   // // TIF[10].FixedLoc : Tool fixed location coded / Emplacement fixe d'outil codé
   // // TIF[11].FixedLoc : Tool fixed location coded / Emplacement fixe d'outil codé
   // // TIF[12].FixedLoc : Tool fixed location coded / Emplacement fixe d'outil codé
   // // TIF[13].FixedLoc : Tool fixed location coded / Emplacement fixe d'outil codé
   // // TIF[14].FixedLoc : Tool fixed location coded / Emplacement fixe d'outil codé
   // // TIF[15].FixedLoc : Tool fixed location coded / Emplacement fixe d'outil codé
   // // TIF[16].FixedLoc : Tool fixed location coded / Emplacement fixe d'outil codé
   // // TIF[2].Used : Tool was in use / Outil a été utilisé
   // // TIF[3].Used : Tool was in use / Outil a été utilisé
   // // TIF[4].Used : Tool was in use / Outil a été utilisé
   // // TIF[5].Used : Tool was in use / Outil a été utilisé
   // // TIF[6].Used : Tool was in use / Outil a été utilisé
   // // TIF[7].Used : Tool was in use / Outil a été utilisé
   // // TIF[8].Used : Tool was in use / Outil a été utilisé
   // // TIF[9].Used : Tool was in use / Outil a été utilisé
   // // TIF[10].Used : Tool was in use / Outil a été utilisé
   // // TIF[11].Used : Tool was in use / Outil a été utilisé
   // // TIF[12].Used : Tool was in use / Outil a été utilisé
   // // TIF[13].Used : Tool was in use / Outil a été utilisé
   // // TIF[14].Used : Tool was in use / Outil a été utilisé
   // // TIF[15].Used : Tool was in use / Outil a été utilisé
   // // TIF[16].Used : Tool was in use / Outil a été utilisé
   // // TIF[2].TNo : Tool new: T number / Nouvel outil : numéro d'outil
   // // TIF[3].TNo : Tool new: T number / Nouvel outil : numéro d'outil
   // // TIF[4].TNo : Tool new: T number / Nouvel outil : numéro d'outil
   // // TIF[5].TNo : Tool new: T number / Nouvel outil : numéro d'outil
   // // TIF[6].TNo : Tool new: T number / Nouvel outil : numéro d'outil
   // // TIF[7].TNo : Tool new: T number / Nouvel outil : numéro d'outil
   // // TIF[8].TNo : Tool new: T number / Nouvel outil : numéro d'outil
   // // TIF[9].TNo : Tool new: T number / Nouvel outil : numéro d'outil
   // // TIF[10].TNo : Tool new: T number / Nouvel outil : numéro d'outil
   // // TIF[11].TNo : Tool new: T number / Nouvel outil : numéro d'outil
   // // TIF[12].TNo : Tool new: T number / Nouvel outil : numéro d'outil
   // // TIF[13].TNo : Tool new: T number / Nouvel outil : numéro d'outil
   // // TIF[14].TNo : Tool new: T number / Nouvel outil : numéro d'outil
   // // TIF[15].TNo : Tool new: T number / Nouvel outil : numéro d'outil
   // // TIF[16].TNo : Tool new: T number / Nouvel outil : numéro d'outil
   // // TIF[2].MyPlace : Original location of new tool / Emplacement d'origine du nouvel outil
   // // TIF[3].MyPlace : Original location of new tool / Emplacement d'origine du nouvel outil
   // // TIF[4].MyPlace : Original location of new tool / Emplacement d'origine du nouvel outil
   // // TIF[5].MyPlace : Original location of new tool / Emplacement d'origine du nouvel outil
   // // TIF[6].MyPlace : Original location of new tool / Emplacement d'origine du nouvel outil
   // // TIF[7].MyPlace : Original location of new tool / Emplacement d'origine du nouvel outil
   // // TIF[8].MyPlace : Original location of new tool / Emplacement d'origine du nouvel outil
   // // TIF[9].MyPlace : Original location of new tool / Emplacement d'origine du nouvel outil
   // // TIF[10].MyPlace : Original location of new tool / Emplacement d'origine du nouvel outil
   // // TIF[11].MyPlace : Original location of new tool / Emplacement d'origine du nouvel outil
   // // TIF[12].MyPlace : Original location of new tool / Emplacement d'origine du nouvel outil
   // // TIF[13].MyPlace : Original location of new tool / Emplacement d'origine du nouvel outil
   // // TIF[14].MyPlace : Original location of new tool / Emplacement d'origine du nouvel outil
   // // TIF[15].MyPlace : Original location of new tool / Emplacement d'origine du nouvel outil
   // // TIF[16].MyPlace : Original location of new tool / Emplacement d'origine du nouvel outil
END_TYPE

TYPE "LBP_typeTMTurretMT"
TITLE = Tool management / Gestion des outils
// User data type for block LBP_TMTurretMT [DB1073] / Type de données utilisateur pour bloc LBP_TMTurretMT [DB1073]
   STRUCT
      MTIF : Array[1..16] of Struct
         DistanceCoding : Int;   // Type of distance coding ($TC_MTP_KD) / Type de codage de distance ($TC_MTP_KD)
         Places : Int;   // Number of locations of the multitool / Nombre d'emplacements Multitool
         Distance : Real;   // Multitool location distance / Distance de l'emplacement Multitool
         NewMTNo : Int;   // MT-Number new Tool / Numéro MT du nouvel outil
         NewPlace : Int;   // Multitool place number / Numéro d'emplacement Multitool
         OldMTNo : Int;   // MT-Number old Tool / Numéro MT de l'ancien outil
         OldPlace : Int;   // Multitool place number / Numéro d'emplacement Multitool
         LocType : Int;   // Tool new: location type / Nouvel outil : type d'emplacement
         SLeft : Int;   // Tool new: size left / Nouvel outil : taille côté gauche
         SRight : Int;   // Tool new: size right / Nouvel outil : taille côté droit
         STop : Int;   // Tool new: size top / Nouvel outil : taille dessus
         SBottom : Int;   // Tool new: size bottom / Nouvel outil : taille dessous
         TInBuffer : Bool;   // ID for tools in buffer / ID pour outils dans tampon
         IgnoreDisabled : Bool;   // Ignore disabled / Ignorer désactivation
         Unload : Bool;   // To be unloaded / À décharger
         Load : Bool;   // To be loaded / À charger
         MasterTool : Bool;   // Tool is the master tool / L'outil est un outil principal
         n26_5 : Bool;   // Reserved / Réservé
         n26_6 : Bool;   // Reserved / Réservé
         HandTool : Bool;   // Hand tool / Outil manuel
         Active : Bool;   // Active tool / Outil actif
         Enabled : Bool;   // Tool enabled / Outil activé
         Disabled : Bool;   // Tool disabled / Outil désactivé
         Measured : Bool;   // Tool measured / Outil mesuré
         Prewarn : Bool;   // Prewarning limit reached / Seuil de préavis atteint
         Change : Bool;   // Tool being changed / Outil en cours de changement
         FixedLoc : Bool;   // Tool fixed location coded / Emplacement fixe d'outil codé
         Used : Bool;   // Tool was in use / Outil a été utilisé
         TNo : Int;   // Tool new: T number / Nouvel outil : numéro d'outil
         Toolholder : Int;   // Toolholder number as tool compensation reference / Numéro de porte-outil en tant que référence pour la compensation d'outil
         MyMag : Int;   // Multitool number the tool is loaded onto / Numéro Multitool dans lequel l'outil est chargé
         MyPlace : Int;   // Multitool place number / Numéro d'emplacement Multitool
         reserved : Array[1..7] of Int;   // Reserved / Réservé
      END_STRUCT;
   END_STRUCT;
   // // MTIF[2].DistanceCoding : Type of distance coding ($TC_MTP_KD) / Type de codage de distance ($TC_MTP_KD)
   // // MTIF[3].DistanceCoding : Type of distance coding ($TC_MTP_KD) / Type de codage de distance ($TC_MTP_KD)
   // // MTIF[4].DistanceCoding : Type of distance coding ($TC_MTP_KD) / Type de codage de distance ($TC_MTP_KD)
   // // MTIF[5].DistanceCoding : Type of distance coding ($TC_MTP_KD) / Type de codage de distance ($TC_MTP_KD)
   // // MTIF[6].DistanceCoding : Type of distance coding ($TC_MTP_KD) / Type de codage de distance ($TC_MTP_KD)
   // // MTIF[7].DistanceCoding : Type of distance coding ($TC_MTP_KD) / Type de codage de distance ($TC_MTP_KD)
   // // MTIF[8].DistanceCoding : Type of distance coding ($TC_MTP_KD) / Type de codage de distance ($TC_MTP_KD)
   // // MTIF[9].DistanceCoding : Type of distance coding ($TC_MTP_KD) / Type de codage de distance ($TC_MTP_KD)
   // // MTIF[10].DistanceCoding : Type of distance coding ($TC_MTP_KD) / Type de codage de distance ($TC_MTP_KD)
   // // MTIF[11].DistanceCoding : Type of distance coding ($TC_MTP_KD) / Type de codage de distance ($TC_MTP_KD)
   // // MTIF[12].DistanceCoding : Type of distance coding ($TC_MTP_KD) / Type de codage de distance ($TC_MTP_KD)
   // // MTIF[13].DistanceCoding : Type of distance coding ($TC_MTP_KD) / Type de codage de distance ($TC_MTP_KD)
   // // MTIF[14].DistanceCoding : Type of distance coding ($TC_MTP_KD) / Type de codage de distance ($TC_MTP_KD)
   // // MTIF[15].DistanceCoding : Type of distance coding ($TC_MTP_KD) / Type de codage de distance ($TC_MTP_KD)
   // // MTIF[16].DistanceCoding : Type of distance coding ($TC_MTP_KD) / Type de codage de distance ($TC_MTP_KD)
   // // MTIF[2].Places : Number of locations of the multitool / Nombre d'emplacements Multitool
   // // MTIF[3].Places : Number of locations of the multitool / Nombre d'emplacements Multitool
   // // MTIF[4].Places : Number of locations of the multitool / Nombre d'emplacements Multitool
   // // MTIF[5].Places : Number of locations of the multitool / Nombre d'emplacements Multitool
   // // MTIF[6].Places : Number of locations of the multitool / Nombre d'emplacements Multitool
   // // MTIF[7].Places : Number of locations of the multitool / Nombre d'emplacements Multitool
   // // MTIF[8].Places : Number of locations of the multitool / Nombre d'emplacements Multitool
   // // MTIF[9].Places : Number of locations of the multitool / Nombre d'emplacements Multitool
   // // MTIF[10].Places : Number of locations of the multitool / Nombre d'emplacements Multitool
   // // MTIF[11].Places : Number of locations of the multitool / Nombre d'emplacements Multitool
   // // MTIF[12].Places : Number of locations of the multitool / Nombre d'emplacements Multitool
   // // MTIF[13].Places : Number of locations of the multitool / Nombre d'emplacements Multitool
   // // MTIF[14].Places : Number of locations of the multitool / Nombre d'emplacements Multitool
   // // MTIF[15].Places : Number of locations of the multitool / Nombre d'emplacements Multitool
   // // MTIF[16].Places : Number of locations of the multitool / Nombre d'emplacements Multitool
   // // MTIF[2].Distance : Multitool location distance / Distance de l'emplacement Multitool
   // // MTIF[3].Distance : Multitool location distance / Distance de l'emplacement Multitool
   // // MTIF[4].Distance : Multitool location distance / Distance de l'emplacement Multitool
   // // MTIF[5].Distance : Multitool location distance / Distance de l'emplacement Multitool
   // // MTIF[6].Distance : Multitool location distance / Distance de l'emplacement Multitool
   // // MTIF[7].Distance : Multitool location distance / Distance de l'emplacement Multitool
   // // MTIF[8].Distance : Multitool location distance / Distance de l'emplacement Multitool
   // // MTIF[9].Distance : Multitool location distance / Distance de l'emplacement Multitool
   // // MTIF[10].Distance : Multitool location distance / Distance de l'emplacement Multitool
   // // MTIF[11].Distance : Multitool location distance / Distance de l'emplacement Multitool
   // // MTIF[12].Distance : Multitool location distance / Distance de l'emplacement Multitool
   // // MTIF[13].Distance : Multitool location distance / Distance de l'emplacement Multitool
   // // MTIF[14].Distance : Multitool location distance / Distance de l'emplacement Multitool
   // // MTIF[15].Distance : Multitool location distance / Distance de l'emplacement Multitool
   // // MTIF[16].Distance : Multitool location distance / Distance de l'emplacement Multitool
   // // MTIF[2].NewMTNo : MT-Number new Tool / Numéro MT du nouvel outil
   // // MTIF[3].NewMTNo : MT-Number new Tool / Numéro MT du nouvel outil
   // // MTIF[4].NewMTNo : MT-Number new Tool / Numéro MT du nouvel outil
   // // MTIF[5].NewMTNo : MT-Number new Tool / Numéro MT du nouvel outil
   // // MTIF[6].NewMTNo : MT-Number new Tool / Numéro MT du nouvel outil
   // // MTIF[7].NewMTNo : MT-Number new Tool / Numéro MT du nouvel outil
   // // MTIF[8].NewMTNo : MT-Number new Tool / Numéro MT du nouvel outil
   // // MTIF[9].NewMTNo : MT-Number new Tool / Numéro MT du nouvel outil
   // // MTIF[10].NewMTNo : MT-Number new Tool / Numéro MT du nouvel outil
   // // MTIF[11].NewMTNo : MT-Number new Tool / Numéro MT du nouvel outil
   // // MTIF[12].NewMTNo : MT-Number new Tool / Numéro MT du nouvel outil
   // // MTIF[13].NewMTNo : MT-Number new Tool / Numéro MT du nouvel outil
   // // MTIF[14].NewMTNo : MT-Number new Tool / Numéro MT du nouvel outil
   // // MTIF[15].NewMTNo : MT-Number new Tool / Numéro MT du nouvel outil
   // // MTIF[16].NewMTNo : MT-Number new Tool / Numéro MT du nouvel outil
   // // MTIF[2].NewPlace : Multitool place number / Numéro d'emplacement Multitool
   // // MTIF[3].NewPlace : Multitool place number / Numéro d'emplacement Multitool
   // // MTIF[4].NewPlace : Multitool place number / Numéro d'emplacement Multitool
   // // MTIF[5].NewPlace : Multitool place number / Numéro d'emplacement Multitool
   // // MTIF[6].NewPlace : Multitool place number / Numéro d'emplacement Multitool
   // // MTIF[7].NewPlace : Multitool place number / Numéro d'emplacement Multitool
   // // MTIF[8].NewPlace : Multitool place number / Numéro d'emplacement Multitool
   // // MTIF[9].NewPlace : Multitool place number / Numéro d'emplacement Multitool
   // // MTIF[10].NewPlace : Multitool place number / Numéro d'emplacement Multitool
   // // MTIF[11].NewPlace : Multitool place number / Numéro d'emplacement Multitool
   // // MTIF[12].NewPlace : Multitool place number / Numéro d'emplacement Multitool
   // // MTIF[13].NewPlace : Multitool place number / Numéro d'emplacement Multitool
   // // MTIF[14].NewPlace : Multitool place number / Numéro d'emplacement Multitool
   // // MTIF[15].NewPlace : Multitool place number / Numéro d'emplacement Multitool
   // // MTIF[16].NewPlace : Multitool place number / Numéro d'emplacement Multitool
   // // MTIF[2].OldMTNo : MT-Number old Tool / Numéro MT de l'ancien outil
   // // MTIF[3].OldMTNo : MT-Number old Tool / Numéro MT de l'ancien outil
   // // MTIF[4].OldMTNo : MT-Number old Tool / Numéro MT de l'ancien outil
   // // MTIF[5].OldMTNo : MT-Number old Tool / Numéro MT de l'ancien outil
   // // MTIF[6].OldMTNo : MT-Number old Tool / Numéro MT de l'ancien outil
   // // MTIF[7].OldMTNo : MT-Number old Tool / Numéro MT de l'ancien outil
   // // MTIF[8].OldMTNo : MT-Number old Tool / Numéro MT de l'ancien outil
   // // MTIF[9].OldMTNo : MT-Number old Tool / Numéro MT de l'ancien outil
   // // MTIF[10].OldMTNo : MT-Number old Tool / Numéro MT de l'ancien outil
   // // MTIF[11].OldMTNo : MT-Number old Tool / Numéro MT de l'ancien outil
   // // MTIF[12].OldMTNo : MT-Number old Tool / Numéro MT de l'ancien outil
   // // MTIF[13].OldMTNo : MT-Number old Tool / Numéro MT de l'ancien outil
   // // MTIF[14].OldMTNo : MT-Number old Tool / Numéro MT de l'ancien outil
   // // MTIF[15].OldMTNo : MT-Number old Tool / Numéro MT de l'ancien outil
   // // MTIF[16].OldMTNo : MT-Number old Tool / Numéro MT de l'ancien outil
   // // MTIF[2].OldPlace : Multitool place number / Numéro d'emplacement Multitool
   // // MTIF[3].OldPlace : Multitool place number / Numéro d'emplacement Multitool
   // // MTIF[4].OldPlace : Multitool place number / Numéro d'emplacement Multitool
   // // MTIF[5].OldPlace : Multitool place number / Numéro d'emplacement Multitool
   // // MTIF[6].OldPlace : Multitool place number / Numéro d'emplacement Multitool
   // // MTIF[7].OldPlace : Multitool place number / Numéro d'emplacement Multitool
   // // MTIF[8].OldPlace : Multitool place number / Numéro d'emplacement Multitool
   // // MTIF[9].OldPlace : Multitool place number / Numéro d'emplacement Multitool
   // // MTIF[10].OldPlace : Multitool place number / Numéro d'emplacement Multitool
   // // MTIF[11].OldPlace : Multitool place number / Numéro d'emplacement Multitool
   // // MTIF[12].OldPlace : Multitool place number / Numéro d'emplacement Multitool
   // // MTIF[13].OldPlace : Multitool place number / Numéro d'emplacement Multitool
   // // MTIF[14].OldPlace : Multitool place number / Numéro d'emplacement Multitool
   // // MTIF[15].OldPlace : Multitool place number / Numéro d'emplacement Multitool
   // // MTIF[16].OldPlace : Multitool place number / Numéro d'emplacement Multitool
   // // MTIF[2].LocType : Tool new: location type / Nouvel outil : type d'emplacement
   // // MTIF[3].LocType : Tool new: location type / Nouvel outil : type d'emplacement
   // // MTIF[4].LocType : Tool new: location type / Nouvel outil : type d'emplacement
   // // MTIF[5].LocType : Tool new: location type / Nouvel outil : type d'emplacement
   // // MTIF[6].LocType : Tool new: location type / Nouvel outil : type d'emplacement
   // // MTIF[7].LocType : Tool new: location type / Nouvel outil : type d'emplacement
   // // MTIF[8].LocType : Tool new: location type / Nouvel outil : type d'emplacement
   // // MTIF[9].LocType : Tool new: location type / Nouvel outil : type d'emplacement
   // // MTIF[10].LocType : Tool new: location type / Nouvel outil : type d'emplacement
   // // MTIF[11].LocType : Tool new: location type / Nouvel outil : type d'emplacement
   // // MTIF[12].LocType : Tool new: location type / Nouvel outil : type d'emplacement
   // // MTIF[13].LocType : Tool new: location type / Nouvel outil : type d'emplacement
   // // MTIF[14].LocType : Tool new: location type / Nouvel outil : type d'emplacement
   // // MTIF[15].LocType : Tool new: location type / Nouvel outil : type d'emplacement
   // // MTIF[16].LocType : Tool new: location type / Nouvel outil : type d'emplacement
   // // MTIF[2].SLeft : Tool new: size left / Nouvel outil : taille côté gauche
   // // MTIF[3].SLeft : Tool new: size left / Nouvel outil : taille côté gauche
   // // MTIF[4].SLeft : Tool new: size left / Nouvel outil : taille côté gauche
   // // MTIF[5].SLeft : Tool new: size left / Nouvel outil : taille côté gauche
   // // MTIF[6].SLeft : Tool new: size left / Nouvel outil : taille côté gauche
   // // MTIF[7].SLeft : Tool new: size left / Nouvel outil : taille côté gauche
   // // MTIF[8].SLeft : Tool new: size left / Nouvel outil : taille côté gauche
   // // MTIF[9].SLeft : Tool new: size left / Nouvel outil : taille côté gauche
   // // MTIF[10].SLeft : Tool new: size left / Nouvel outil : taille côté gauche
   // // MTIF[11].SLeft : Tool new: size left / Nouvel outil : taille côté gauche
   // // MTIF[12].SLeft : Tool new: size left / Nouvel outil : taille côté gauche
   // // MTIF[13].SLeft : Tool new: size left / Nouvel outil : taille côté gauche
   // // MTIF[14].SLeft : Tool new: size left / Nouvel outil : taille côté gauche
   // // MTIF[15].SLeft : Tool new: size left / Nouvel outil : taille côté gauche
   // // MTIF[16].SLeft : Tool new: size left / Nouvel outil : taille côté gauche
   // // MTIF[2].SRight : Tool new: size right / Nouvel outil : taille côté droit
   // // MTIF[3].SRight : Tool new: size right / Nouvel outil : taille côté droit
   // // MTIF[4].SRight : Tool new: size right / Nouvel outil : taille côté droit
   // // MTIF[5].SRight : Tool new: size right / Nouvel outil : taille côté droit
   // // MTIF[6].SRight : Tool new: size right / Nouvel outil : taille côté droit
   // // MTIF[7].SRight : Tool new: size right / Nouvel outil : taille côté droit
   // // MTIF[8].SRight : Tool new: size right / Nouvel outil : taille côté droit
   // // MTIF[9].SRight : Tool new: size right / Nouvel outil : taille côté droit
   // // MTIF[10].SRight : Tool new: size right / Nouvel outil : taille côté droit
   // // MTIF[11].SRight : Tool new: size right / Nouvel outil : taille côté droit
   // // MTIF[12].SRight : Tool new: size right / Nouvel outil : taille côté droit
   // // MTIF[13].SRight : Tool new: size right / Nouvel outil : taille côté droit
   // // MTIF[14].SRight : Tool new: size right / Nouvel outil : taille côté droit
   // // MTIF[15].SRight : Tool new: size right / Nouvel outil : taille côté droit
   // // MTIF[16].SRight : Tool new: size right / Nouvel outil : taille côté droit
   // // MTIF[2].STop : Tool new: size top / Nouvel outil : taille dessus
   // // MTIF[3].STop : Tool new: size top / Nouvel outil : taille dessus
   // // MTIF[4].STop : Tool new: size top / Nouvel outil : taille dessus
   // // MTIF[5].STop : Tool new: size top / Nouvel outil : taille dessus
   // // MTIF[6].STop : Tool new: size top / Nouvel outil : taille dessus
   // // MTIF[7].STop : Tool new: size top / Nouvel outil : taille dessus
   // // MTIF[8].STop : Tool new: size top / Nouvel outil : taille dessus
   // // MTIF[9].STop : Tool new: size top / Nouvel outil : taille dessus
   // // MTIF[10].STop : Tool new: size top / Nouvel outil : taille dessus
   // // MTIF[11].STop : Tool new: size top / Nouvel outil : taille dessus
   // // MTIF[12].STop : Tool new: size top / Nouvel outil : taille dessus
   // // MTIF[13].STop : Tool new: size top / Nouvel outil : taille dessus
   // // MTIF[14].STop : Tool new: size top / Nouvel outil : taille dessus
   // // MTIF[15].STop : Tool new: size top / Nouvel outil : taille dessus
   // // MTIF[16].STop : Tool new: size top / Nouvel outil : taille dessus
   // // MTIF[2].SBottom : Tool new: size bottom / Nouvel outil : taille dessous
   // // MTIF[3].SBottom : Tool new: size bottom / Nouvel outil : taille dessous
   // // MTIF[4].SBottom : Tool new: size bottom / Nouvel outil : taille dessous
   // // MTIF[5].SBottom : Tool new: size bottom / Nouvel outil : taille dessous
   // // MTIF[6].SBottom : Tool new: size bottom / Nouvel outil : taille dessous
   // // MTIF[7].SBottom : Tool new: size bottom / Nouvel outil : taille dessous
   // // MTIF[8].SBottom : Tool new: size bottom / Nouvel outil : taille dessous
   // // MTIF[9].SBottom : Tool new: size bottom / Nouvel outil : taille dessous
   // // MTIF[10].SBottom : Tool new: size bottom / Nouvel outil : taille dessous
   // // MTIF[11].SBottom : Tool new: size bottom / Nouvel outil : taille dessous
   // // MTIF[12].SBottom : Tool new: size bottom / Nouvel outil : taille dessous
   // // MTIF[13].SBottom : Tool new: size bottom / Nouvel outil : taille dessous
   // // MTIF[14].SBottom : Tool new: size bottom / Nouvel outil : taille dessous
   // // MTIF[15].SBottom : Tool new: size bottom / Nouvel outil : taille dessous
   // // MTIF[16].SBottom : Tool new: size bottom / Nouvel outil : taille dessous
   // // MTIF[2].TInBuffer : ID for tools in buffer / ID pour outils dans tampon
   // // MTIF[3].TInBuffer : ID for tools in buffer / ID pour outils dans tampon
   // // MTIF[4].TInBuffer : ID for tools in buffer / ID pour outils dans tampon
   // // MTIF[5].TInBuffer : ID for tools in buffer / ID pour outils dans tampon
   // // MTIF[6].TInBuffer : ID for tools in buffer / ID pour outils dans tampon
   // // MTIF[7].TInBuffer : ID for tools in buffer / ID pour outils dans tampon
   // // MTIF[8].TInBuffer : ID for tools in buffer / ID pour outils dans tampon
   // // MTIF[9].TInBuffer : ID for tools in buffer / ID pour outils dans tampon
   // // MTIF[10].TInBuffer : ID for tools in buffer / ID pour outils dans tampon
   // // MTIF[11].TInBuffer : ID for tools in buffer / ID pour outils dans tampon
   // // MTIF[12].TInBuffer : ID for tools in buffer / ID pour outils dans tampon
   // // MTIF[13].TInBuffer : ID for tools in buffer / ID pour outils dans tampon
   // // MTIF[14].TInBuffer : ID for tools in buffer / ID pour outils dans tampon
   // // MTIF[15].TInBuffer : ID for tools in buffer / ID pour outils dans tampon
   // // MTIF[16].TInBuffer : ID for tools in buffer / ID pour outils dans tampon
   // // MTIF[2].IgnoreDisabled : Ignore disabled / Ignorer désactivation
   // // MTIF[3].IgnoreDisabled : Ignore disabled / Ignorer désactivation
   // // MTIF[4].IgnoreDisabled : Ignore disabled / Ignorer désactivation
   // // MTIF[5].IgnoreDisabled : Ignore disabled / Ignorer désactivation
   // // MTIF[6].IgnoreDisabled : Ignore disabled / Ignorer désactivation
   // // MTIF[7].IgnoreDisabled : Ignore disabled / Ignorer désactivation
   // // MTIF[8].IgnoreDisabled : Ignore disabled / Ignorer désactivation
   // // MTIF[9].IgnoreDisabled : Ignore disabled / Ignorer désactivation
   // // MTIF[10].IgnoreDisabled : Ignore disabled / Ignorer désactivation
   // // MTIF[11].IgnoreDisabled : Ignore disabled / Ignorer désactivation
   // // MTIF[12].IgnoreDisabled : Ignore disabled / Ignorer désactivation
   // // MTIF[13].IgnoreDisabled : Ignore disabled / Ignorer désactivation
   // // MTIF[14].IgnoreDisabled : Ignore disabled / Ignorer désactivation
   // // MTIF[15].IgnoreDisabled : Ignore disabled / Ignorer désactivation
   // // MTIF[16].IgnoreDisabled : Ignore disabled / Ignorer désactivation
   // // MTIF[2].Unload : To be unloaded / À décharger
   // // MTIF[3].Unload : To be unloaded / À décharger
   // // MTIF[4].Unload : To be unloaded / À décharger
   // // MTIF[5].Unload : To be unloaded / À décharger
   // // MTIF[6].Unload : To be unloaded / À décharger
   // // MTIF[7].Unload : To be unloaded / À décharger
   // // MTIF[8].Unload : To be unloaded / À décharger
   // // MTIF[9].Unload : To be unloaded / À décharger
   // // MTIF[10].Unload : To be unloaded / À décharger
   // // MTIF[11].Unload : To be unloaded / À décharger
   // // MTIF[12].Unload : To be unloaded / À décharger
   // // MTIF[13].Unload : To be unloaded / À décharger
   // // MTIF[14].Unload : To be unloaded / À décharger
   // // MTIF[15].Unload : To be unloaded / À décharger
   // // MTIF[16].Unload : To be unloaded / À décharger
   // // MTIF[2].Load : To be loaded / À charger
   // // MTIF[3].Load : To be loaded / À charger
   // // MTIF[4].Load : To be loaded / À charger
   // // MTIF[5].Load : To be loaded / À charger
   // // MTIF[6].Load : To be loaded / À charger
   // // MTIF[7].Load : To be loaded / À charger
   // // MTIF[8].Load : To be loaded / À charger
   // // MTIF[9].Load : To be loaded / À charger
   // // MTIF[10].Load : To be loaded / À charger
   // // MTIF[11].Load : To be loaded / À charger
   // // MTIF[12].Load : To be loaded / À charger
   // // MTIF[13].Load : To be loaded / À charger
   // // MTIF[14].Load : To be loaded / À charger
   // // MTIF[15].Load : To be loaded / À charger
   // // MTIF[16].Load : To be loaded / À charger
   // // MTIF[2].MasterTool : Tool is the master tool / L'outil est un outil principal
   // // MTIF[3].MasterTool : Tool is the master tool / L'outil est un outil principal
   // // MTIF[4].MasterTool : Tool is the master tool / L'outil est un outil principal
   // // MTIF[5].MasterTool : Tool is the master tool / L'outil est un outil principal
   // // MTIF[6].MasterTool : Tool is the master tool / L'outil est un outil principal
   // // MTIF[7].MasterTool : Tool is the master tool / L'outil est un outil principal
   // // MTIF[8].MasterTool : Tool is the master tool / L'outil est un outil principal
   // // MTIF[9].MasterTool : Tool is the master tool / L'outil est un outil principal
   // // MTIF[10].MasterTool : Tool is the master tool / L'outil est un outil principal
   // // MTIF[11].MasterTool : Tool is the master tool / L'outil est un outil principal
   // // MTIF[12].MasterTool : Tool is the master tool / L'outil est un outil principal
   // // MTIF[13].MasterTool : Tool is the master tool / L'outil est un outil principal
   // // MTIF[14].MasterTool : Tool is the master tool / L'outil est un outil principal
   // // MTIF[15].MasterTool : Tool is the master tool / L'outil est un outil principal
   // // MTIF[16].MasterTool : Tool is the master tool / L'outil est un outil principal
   // // MTIF[2].n26_5 : Reserved / Réservé
   // // MTIF[3].n26_5 : Reserved / Réservé
   // // MTIF[4].n26_5 : Reserved / Réservé
   // // MTIF[5].n26_5 : Reserved / Réservé
   // // MTIF[6].n26_5 : Reserved / Réservé
   // // MTIF[7].n26_5 : Reserved / Réservé
   // // MTIF[8].n26_5 : Reserved / Réservé
   // // MTIF[9].n26_5 : Reserved / Réservé
   // // MTIF[10].n26_5 : Reserved / Réservé
   // // MTIF[11].n26_5 : Reserved / Réservé
   // // MTIF[12].n26_5 : Reserved / Réservé
   // // MTIF[13].n26_5 : Reserved / Réservé
   // // MTIF[14].n26_5 : Reserved / Réservé
   // // MTIF[15].n26_5 : Reserved / Réservé
   // // MTIF[16].n26_5 : Reserved / Réservé
   // // MTIF[2].n26_6 : Reserved / Réservé
   // // MTIF[3].n26_6 : Reserved / Réservé
   // // MTIF[4].n26_6 : Reserved / Réservé
   // // MTIF[5].n26_6 : Reserved / Réservé
   // // MTIF[6].n26_6 : Reserved / Réservé
   // // MTIF[7].n26_6 : Reserved / Réservé
   // // MTIF[8].n26_6 : Reserved / Réservé
   // // MTIF[9].n26_6 : Reserved / Réservé
   // // MTIF[10].n26_6 : Reserved / Réservé
   // // MTIF[11].n26_6 : Reserved / Réservé
   // // MTIF[12].n26_6 : Reserved / Réservé
   // // MTIF[13].n26_6 : Reserved / Réservé
   // // MTIF[14].n26_6 : Reserved / Réservé
   // // MTIF[15].n26_6 : Reserved / Réservé
   // // MTIF[16].n26_6 : Reserved / Réservé
   // // MTIF[2].HandTool : Hand tool / Outil manuel
   // // MTIF[3].HandTool : Hand tool / Outil manuel
   // // MTIF[4].HandTool : Hand tool / Outil manuel
   // // MTIF[5].HandTool : Hand tool / Outil manuel
   // // MTIF[6].HandTool : Hand tool / Outil manuel
   // // MTIF[7].HandTool : Hand tool / Outil manuel
   // // MTIF[8].HandTool : Hand tool / Outil manuel
   // // MTIF[9].HandTool : Hand tool / Outil manuel
   // // MTIF[10].HandTool : Hand tool / Outil manuel
   // // MTIF[11].HandTool : Hand tool / Outil manuel
   // // MTIF[12].HandTool : Hand tool / Outil manuel
   // // MTIF[13].HandTool : Hand tool / Outil manuel
   // // MTIF[14].HandTool : Hand tool / Outil manuel
   // // MTIF[15].HandTool : Hand tool / Outil manuel
   // // MTIF[16].HandTool : Hand tool / Outil manuel
   // // MTIF[2].Active : Active tool / Outil actif
   // // MTIF[3].Active : Active tool / Outil actif
   // // MTIF[4].Active : Active tool / Outil actif
   // // MTIF[5].Active : Active tool / Outil actif
   // // MTIF[6].Active : Active tool / Outil actif
   // // MTIF[7].Active : Active tool / Outil actif
   // // MTIF[8].Active : Active tool / Outil actif
   // // MTIF[9].Active : Active tool / Outil actif
   // // MTIF[10].Active : Active tool / Outil actif
   // // MTIF[11].Active : Active tool / Outil actif
   // // MTIF[12].Active : Active tool / Outil actif
   // // MTIF[13].Active : Active tool / Outil actif
   // // MTIF[14].Active : Active tool / Outil actif
   // // MTIF[15].Active : Active tool / Outil actif
   // // MTIF[16].Active : Active tool / Outil actif
   // // MTIF[2].Enabled : Tool enabled / Outil activé
   // // MTIF[3].Enabled : Tool enabled / Outil activé
   // // MTIF[4].Enabled : Tool enabled / Outil activé
   // // MTIF[5].Enabled : Tool enabled / Outil activé
   // // MTIF[6].Enabled : Tool enabled / Outil activé
   // // MTIF[7].Enabled : Tool enabled / Outil activé
   // // MTIF[8].Enabled : Tool enabled / Outil activé
   // // MTIF[9].Enabled : Tool enabled / Outil activé
   // // MTIF[10].Enabled : Tool enabled / Outil activé
   // // MTIF[11].Enabled : Tool enabled / Outil activé
   // // MTIF[12].Enabled : Tool enabled / Outil activé
   // // MTIF[13].Enabled : Tool enabled / Outil activé
   // // MTIF[14].Enabled : Tool enabled / Outil activé
   // // MTIF[15].Enabled : Tool enabled / Outil activé
   // // MTIF[16].Enabled : Tool enabled / Outil activé
   // // MTIF[2].Disabled : Tool disabled / Outil désactivé
   // // MTIF[3].Disabled : Tool disabled / Outil désactivé
   // // MTIF[4].Disabled : Tool disabled / Outil désactivé
   // // MTIF[5].Disabled : Tool disabled / Outil désactivé
   // // MTIF[6].Disabled : Tool disabled / Outil désactivé
   // // MTIF[7].Disabled : Tool disabled / Outil désactivé
   // // MTIF[8].Disabled : Tool disabled / Outil désactivé
   // // MTIF[9].Disabled : Tool disabled / Outil désactivé
   // // MTIF[10].Disabled : Tool disabled / Outil désactivé
   // // MTIF[11].Disabled : Tool disabled / Outil désactivé
   // // MTIF[12].Disabled : Tool disabled / Outil désactivé
   // // MTIF[13].Disabled : Tool disabled / Outil désactivé
   // // MTIF[14].Disabled : Tool disabled / Outil désactivé
   // // MTIF[15].Disabled : Tool disabled / Outil désactivé
   // // MTIF[16].Disabled : Tool disabled / Outil désactivé
   // // MTIF[2].Measured : Tool measured / Outil mesuré
   // // MTIF[3].Measured : Tool measured / Outil mesuré
   // // MTIF[4].Measured : Tool measured / Outil mesuré
   // // MTIF[5].Measured : Tool measured / Outil mesuré
   // // MTIF[6].Measured : Tool measured / Outil mesuré
   // // MTIF[7].Measured : Tool measured / Outil mesuré
   // // MTIF[8].Measured : Tool measured / Outil mesuré
   // // MTIF[9].Measured : Tool measured / Outil mesuré
   // // MTIF[10].Measured : Tool measured / Outil mesuré
   // // MTIF[11].Measured : Tool measured / Outil mesuré
   // // MTIF[12].Measured : Tool measured / Outil mesuré
   // // MTIF[13].Measured : Tool measured / Outil mesuré
   // // MTIF[14].Measured : Tool measured / Outil mesuré
   // // MTIF[15].Measured : Tool measured / Outil mesuré
   // // MTIF[16].Measured : Tool measured / Outil mesuré
   // // MTIF[2].Prewarn : Prewarning limit reached / Seuil de préavis atteint
   // // MTIF[3].Prewarn : Prewarning limit reached / Seuil de préavis atteint
   // // MTIF[4].Prewarn : Prewarning limit reached / Seuil de préavis atteint
   // // MTIF[5].Prewarn : Prewarning limit reached / Seuil de préavis atteint
   // // MTIF[6].Prewarn : Prewarning limit reached / Seuil de préavis atteint
   // // MTIF[7].Prewarn : Prewarning limit reached / Seuil de préavis atteint
   // // MTIF[8].Prewarn : Prewarning limit reached / Seuil de préavis atteint
   // // MTIF[9].Prewarn : Prewarning limit reached / Seuil de préavis atteint
   // // MTIF[10].Prewarn : Prewarning limit reached / Seuil de préavis atteint
   // // MTIF[11].Prewarn : Prewarning limit reached / Seuil de préavis atteint
   // // MTIF[12].Prewarn : Prewarning limit reached / Seuil de préavis atteint
   // // MTIF[13].Prewarn : Prewarning limit reached / Seuil de préavis atteint
   // // MTIF[14].Prewarn : Prewarning limit reached / Seuil de préavis atteint
   // // MTIF[15].Prewarn : Prewarning limit reached / Seuil de préavis atteint
   // // MTIF[16].Prewarn : Prewarning limit reached / Seuil de préavis atteint
   // // MTIF[2].Change : Tool being changed / Outil en cours de changement
   // // MTIF[3].Change : Tool being changed / Outil en cours de changement
   // // MTIF[4].Change : Tool being changed / Outil en cours de changement
   // // MTIF[5].Change : Tool being changed / Outil en cours de changement
   // // MTIF[6].Change : Tool being changed / Outil en cours de changement
   // // MTIF[7].Change : Tool being changed / Outil en cours de changement
   // // MTIF[8].Change : Tool being changed / Outil en cours de changement
   // // MTIF[9].Change : Tool being changed / Outil en cours de changement
   // // MTIF[10].Change : Tool being changed / Outil en cours de changement
   // // MTIF[11].Change : Tool being changed / Outil en cours de changement
   // // MTIF[12].Change : Tool being changed / Outil en cours de changement
   // // MTIF[13].Change : Tool being changed / Outil en cours de changement
   // // MTIF[14].Change : Tool being changed / Outil en cours de changement
   // // MTIF[15].Change : Tool being changed / Outil en cours de changement
   // // MTIF[16].Change : Tool being changed / Outil en cours de changement
   // // MTIF[2].FixedLoc : Tool fixed location coded / Emplacement fixe d'outil codé
   // // MTIF[3].FixedLoc : Tool fixed location coded / Emplacement fixe d'outil codé
   // // MTIF[4].FixedLoc : Tool fixed location coded / Emplacement fixe d'outil codé
   // // MTIF[5].FixedLoc : Tool fixed location coded / Emplacement fixe d'outil codé
   // // MTIF[6].FixedLoc : Tool fixed location coded / Emplacement fixe d'outil codé
   // // MTIF[7].FixedLoc : Tool fixed location coded / Emplacement fixe d'outil codé
   // // MTIF[8].FixedLoc : Tool fixed location coded / Emplacement fixe d'outil codé
   // // MTIF[9].FixedLoc : Tool fixed location coded / Emplacement fixe d'outil codé
   // // MTIF[10].FixedLoc : Tool fixed location coded / Emplacement fixe d'outil codé
   // // MTIF[11].FixedLoc : Tool fixed location coded / Emplacement fixe d'outil codé
   // // MTIF[12].FixedLoc : Tool fixed location coded / Emplacement fixe d'outil codé
   // // MTIF[13].FixedLoc : Tool fixed location coded / Emplacement fixe d'outil codé
   // // MTIF[14].FixedLoc : Tool fixed location coded / Emplacement fixe d'outil codé
   // // MTIF[15].FixedLoc : Tool fixed location coded / Emplacement fixe d'outil codé
   // // MTIF[16].FixedLoc : Tool fixed location coded / Emplacement fixe d'outil codé
   // // MTIF[2].Used : Tool was in use / Outil a été utilisé
   // // MTIF[3].Used : Tool was in use / Outil a été utilisé
   // // MTIF[4].Used : Tool was in use / Outil a été utilisé
   // // MTIF[5].Used : Tool was in use / Outil a été utilisé
   // // MTIF[6].Used : Tool was in use / Outil a été utilisé
   // // MTIF[7].Used : Tool was in use / Outil a été utilisé
   // // MTIF[8].Used : Tool was in use / Outil a été utilisé
   // // MTIF[9].Used : Tool was in use / Outil a été utilisé
   // // MTIF[10].Used : Tool was in use / Outil a été utilisé
   // // MTIF[11].Used : Tool was in use / Outil a été utilisé
   // // MTIF[12].Used : Tool was in use / Outil a été utilisé
   // // MTIF[13].Used : Tool was in use / Outil a été utilisé
   // // MTIF[14].Used : Tool was in use / Outil a été utilisé
   // // MTIF[15].Used : Tool was in use / Outil a été utilisé
   // // MTIF[16].Used : Tool was in use / Outil a été utilisé
   // // MTIF[2].TNo : Tool new: T number / Nouvel outil : numéro d'outil
   // // MTIF[3].TNo : Tool new: T number / Nouvel outil : numéro d'outil
   // // MTIF[4].TNo : Tool new: T number / Nouvel outil : numéro d'outil
   // // MTIF[5].TNo : Tool new: T number / Nouvel outil : numéro d'outil
   // // MTIF[6].TNo : Tool new: T number / Nouvel outil : numéro d'outil
   // // MTIF[7].TNo : Tool new: T number / Nouvel outil : numéro d'outil
   // // MTIF[8].TNo : Tool new: T number / Nouvel outil : numéro d'outil
   // // MTIF[9].TNo : Tool new: T number / Nouvel outil : numéro d'outil
   // // MTIF[10].TNo : Tool new: T number / Nouvel outil : numéro d'outil
   // // MTIF[11].TNo : Tool new: T number / Nouvel outil : numéro d'outil
   // // MTIF[12].TNo : Tool new: T number / Nouvel outil : numéro d'outil
   // // MTIF[13].TNo : Tool new: T number / Nouvel outil : numéro d'outil
   // // MTIF[14].TNo : Tool new: T number / Nouvel outil : numéro d'outil
   // // MTIF[15].TNo : Tool new: T number / Nouvel outil : numéro d'outil
   // // MTIF[16].TNo : Tool new: T number / Nouvel outil : numéro d'outil
   // // MTIF[2].Toolholder : Toolholder number as tool compensation reference / Numéro de porte-outil en tant que référence pour la compensation d'outil
   // // MTIF[3].Toolholder : Toolholder number as tool compensation reference / Numéro de porte-outil en tant que référence pour la compensation d'outil
   // // MTIF[4].Toolholder : Toolholder number as tool compensation reference / Numéro de porte-outil en tant que référence pour la compensation d'outil
   // // MTIF[5].Toolholder : Toolholder number as tool compensation reference / Numéro de porte-outil en tant que référence pour la compensation d'outil
   // // MTIF[6].Toolholder : Toolholder number as tool compensation reference / Numéro de porte-outil en tant que référence pour la compensation d'outil
   // // MTIF[7].Toolholder : Toolholder number as tool compensation reference / Numéro de porte-outil en tant que référence pour la compensation d'outil
   // // MTIF[8].Toolholder : Toolholder number as tool compensation reference / Numéro de porte-outil en tant que référence pour la compensation d'outil
   // // MTIF[9].Toolholder : Toolholder number as tool compensation reference / Numéro de porte-outil en tant que référence pour la compensation d'outil
   // // MTIF[10].Toolholder : Toolholder number as tool compensation reference / Numéro de porte-outil en tant que référence pour la compensation d'outil
   // // MTIF[11].Toolholder : Toolholder number as tool compensation reference / Numéro de porte-outil en tant que référence pour la compensation d'outil
   // // MTIF[12].Toolholder : Toolholder number as tool compensation reference / Numéro de porte-outil en tant que référence pour la compensation d'outil
   // // MTIF[13].Toolholder : Toolholder number as tool compensation reference / Numéro de porte-outil en tant que référence pour la compensation d'outil
   // // MTIF[14].Toolholder : Toolholder number as tool compensation reference / Numéro de porte-outil en tant que référence pour la compensation d'outil
   // // MTIF[15].Toolholder : Toolholder number as tool compensation reference / Numéro de porte-outil en tant que référence pour la compensation d'outil
   // // MTIF[16].Toolholder : Toolholder number as tool compensation reference / Numéro de porte-outil en tant que référence pour la compensation d'outil
   // // MTIF[2].MyMag : Multitool number the tool is loaded onto / Numéro Multitool dans lequel l'outil est chargé
   // // MTIF[3].MyMag : Multitool number the tool is loaded onto / Numéro Multitool dans lequel l'outil est chargé
   // // MTIF[4].MyMag : Multitool number the tool is loaded onto / Numéro Multitool dans lequel l'outil est chargé
   // // MTIF[5].MyMag : Multitool number the tool is loaded onto / Numéro Multitool dans lequel l'outil est chargé
   // // MTIF[6].MyMag : Multitool number the tool is loaded onto / Numéro Multitool dans lequel l'outil est chargé
   // // MTIF[7].MyMag : Multitool number the tool is loaded onto / Numéro Multitool dans lequel l'outil est chargé
   // // MTIF[8].MyMag : Multitool number the tool is loaded onto / Numéro Multitool dans lequel l'outil est chargé
   // // MTIF[9].MyMag : Multitool number the tool is loaded onto / Numéro Multitool dans lequel l'outil est chargé
   // // MTIF[10].MyMag : Multitool number the tool is loaded onto / Numéro Multitool dans lequel l'outil est chargé
   // // MTIF[11].MyMag : Multitool number the tool is loaded onto / Numéro Multitool dans lequel l'outil est chargé
   // // MTIF[12].MyMag : Multitool number the tool is loaded onto / Numéro Multitool dans lequel l'outil est chargé
   // // MTIF[13].MyMag : Multitool number the tool is loaded onto / Numéro Multitool dans lequel l'outil est chargé
   // // MTIF[14].MyMag : Multitool number the tool is loaded onto / Numéro Multitool dans lequel l'outil est chargé
   // // MTIF[15].MyMag : Multitool number the tool is loaded onto / Numéro Multitool dans lequel l'outil est chargé
   // // MTIF[16].MyMag : Multitool number the tool is loaded onto / Numéro Multitool dans lequel l'outil est chargé
   // // MTIF[2].MyPlace : Multitool place number / Numéro d'emplacement Multitool
   // // MTIF[3].MyPlace : Multitool place number / Numéro d'emplacement Multitool
   // // MTIF[4].MyPlace : Multitool place number / Numéro d'emplacement Multitool
   // // MTIF[5].MyPlace : Multitool place number / Numéro d'emplacement Multitool
   // // MTIF[6].MyPlace : Multitool place number / Numéro d'emplacement Multitool
   // // MTIF[7].MyPlace : Multitool place number / Numéro d'emplacement Multitool
   // // MTIF[8].MyPlace : Multitool place number / Numéro d'emplacement Multitool
   // // MTIF[9].MyPlace : Multitool place number / Numéro d'emplacement Multitool
   // // MTIF[10].MyPlace : Multitool place number / Numéro d'emplacement Multitool
   // // MTIF[11].MyPlace : Multitool place number / Numéro d'emplacement Multitool
   // // MTIF[12].MyPlace : Multitool place number / Numéro d'emplacement Multitool
   // // MTIF[13].MyPlace : Multitool place number / Numéro d'emplacement Multitool
   // // MTIF[14].MyPlace : Multitool place number / Numéro d'emplacement Multitool
   // // MTIF[15].MyPlace : Multitool place number / Numéro d'emplacement Multitool
   // // MTIF[16].MyPlace : Multitool place number / Numéro d'emplacement Multitool
   // // MTIF[2].reserved : Reserved / Réservé
   // // MTIF[3].reserved : Reserved / Réservé
   // // MTIF[4].reserved : Reserved / Réservé
   // // MTIF[5].reserved : Reserved / Réservé
   // // MTIF[6].reserved : Reserved / Réservé
   // // MTIF[7].reserved : Reserved / Réservé
   // // MTIF[8].reserved : Reserved / Réservé
   // // MTIF[9].reserved : Reserved / Réservé
   // // MTIF[10].reserved : Reserved / Réservé
   // // MTIF[11].reserved : Reserved / Réservé
   // // MTIF[12].reserved : Reserved / Réservé
   // // MTIF[13].reserved : Reserved / Réservé
   // // MTIF[14].reserved : Reserved / Réservé
   // // MTIF[15].reserved : Reserved / Réservé
   // // MTIF[16].reserved : Reserved / Réservé
END_TYPE

TYPE "DT_DataFromSafety"
// stored: IsFailsafeCompliant true
   STRUCT
      iSafety_EStop { ExternalAccessible := 'False'; ExternalVisible := 'False'; ExternalWritable := 'False'} : Bool;
      iKeySettingMode { ExternalAccessible := 'False'; ExternalVisible := 'False'; ExternalWritable := 'False'} : Bool;
      iKeySettingLaser { ExternalAccessible := 'False'; ExternalVisible := 'False'; ExternalWritable := 'False'} : Bool;
      iBackMachine { ExternalAccessible := 'False'; ExternalVisible := 'False'; ExternalWritable := 'False'} : Bool;
      iBackExternal : Bool;
      iReturnPowerLaser { ExternalAccessible := 'False'; ExternalVisible := 'False'; ExternalWritable := 'False'} : Bool;
      iMaintenanceDoorClosed { ExternalAccessible := 'False'; ExternalVisible := 'False'; ExternalWritable := 'False'} : Bool;
      iFrontDoorClosed { ExternalAccessible := 'False'; ExternalVisible := 'False'; ExternalWritable := 'False'} : Bool;
      iEmergencyStopPowerLaser { ExternalAccessible := 'False'; ExternalVisible := 'False'; ExternalWritable := 'False'} : Bool;
      iReturnShutterLaser { ExternalAccessible := 'False'; ExternalVisible := 'False'; ExternalWritable := 'False'} : Bool;
      iRoofLeftDoorClosed { ExternalAccessible := 'False'; ExternalVisible := 'False'; ExternalWritable := 'False'} : Bool;
      iKeyLaserOn { ExternalAccessible := 'False'; ExternalVisible := 'False'; ExternalWritable := 'False'} : Bool;
      iLaserExternDoorClosed : Bool;
      iSasOneDoorClosed : Bool;
      iBwLoaderDoorClosed : Bool;
      iRoofRightDoorClosed { ExternalAccessible := 'False'; ExternalVisible := 'False'; ExternalWritable := 'False'} : Bool;
      iSonplas_EStop : Bool;
      iBwLoader_EStop : Bool;
      iSonplasDoorClosed : Bool;
      iReturnDoorClosed : Bool;
      oContactorMachine { ExternalAccessible := 'False'; ExternalVisible := 'False'; ExternalWritable := 'False'} : Bool;
      oContactorLaser { ExternalAccessible := 'False'; ExternalVisible := 'False'; ExternalWritable := 'False'} : Bool;
      oContactorShutter { ExternalAccessible := 'False'; ExternalVisible := 'False'; ExternalWritable := 'False'} : Bool;
      oBwLoaderEStopRelay : Bool;
      oSonplasDoorClosedRelay : Bool;
      EmergencyStop { ExternalAccessible := 'False'; ExternalVisible := 'False'; ExternalWritable := 'False'} : Bool;
      DoorsClosed { ExternalAccessible := 'False'; ExternalVisible := 'False'; ExternalWritable := 'False'} : Bool;
      ModeSettingLaser { ExternalAccessible := 'False'; ExternalVisible := 'False'; ExternalWritable := 'False'} : Bool;
      ShutterClosed { ExternalAccessible := 'False'; ExternalVisible := 'False'; ExternalWritable := 'False'} : Bool;
      ShutterReadyToOpen { ExternalAccessible := 'False'; ExternalVisible := 'False'; ExternalWritable := 'False'} : Bool;
      ShutterOpened { ExternalAccessible := 'False'; ExternalVisible := 'False'; ExternalWritable := 'False'} : Bool;
      ShutterError { ExternalAccessible := 'False'; ExternalVisible := 'False'; ExternalWritable := 'False'} : Bool;
      LaserSupplyPowerError { ExternalAccessible := 'False'; ExternalVisible := 'False'; ExternalWritable := 'False'} : Bool;
      SupplyPowerError { ExternalAccessible := 'False'; ExternalVisible := 'False'; ExternalWritable := 'False'} : Bool;
      BW_LoaderEstopRelayError : Bool;
      SonplasDoorClosedRelayError : Bool;
      Comissionning { ExternalAccessible := 'False'; ExternalVisible := 'False'; ExternalWritable := 'False'} : Bool;
      OpenShutter { ExternalAccessible := 'False'; ExternalVisible := 'False'; ExternalWritable := 'False'} : Bool;
      AllDoorLockedForLaser { ExternalAccessible := 'False'; ExternalVisible := 'False'; ExternalWritable := 'False'} : Bool;
      AckEmergencyStop { ExternalAccessible := 'False'; ExternalVisible := 'False'; ExternalWritable := 'False'} : Bool;
      AckFdbPowLaser { ExternalAccessible := 'False'; ExternalVisible := 'False'; ExternalWritable := 'False'} : Bool;
      AckI2001Functions { ExternalAccessible := 'False'; ExternalVisible := 'False'; ExternalWritable := 'False'} : Bool;
   END_STRUCT;
END_TYPE

TYPE "DT_DataToSafety"
// stored: IsFailsafeCompliant true
   STRUCT
      OpenShutterButton : Bool;
      ResetEmergencyStop : Bool;
      JOG_Mod : Bool;
      Activation_Axis : Bool;
      CloseShutter : Bool;
      FrontDoorLock : Bool;
      DoorsInhibit : Bool;
   END_STRUCT;
END_TYPE

TYPE "LBP_typeHandwheel"
TITLE = Handwheel image / Image de la manivelle
// User data type for handwheel / Type de données utilisateur pour manivelle
   STRUCT
      handWheel1 : Int;
      handWheel2 : Int;
   END_STRUCT;
END_TYPE

TYPE "LBP_typeMcp310AdditionalInput"
TITLE = MCP 310 image / Image du MCP 310
// Additional input image of MCP 310 / Image d'entrée supplémentaire du MCP 310
   STRUCT
      directKey1 : Bool;   // DT1
      directKey2 : Bool;   // DT2
      directKey3 : Bool;   // DT3
      directKey4 : Bool;   // DT4
      directKey5 : Bool;   // DT5
      directKey6 : Bool;   // DT6
      directKey7 : Bool;   // DT7
      directKey8 : Bool;   // DT8
      directKey9 : Bool;   // DT9
      directKey10 : Bool;   // DT10
      directKey11 : Bool;   // DT11
      directKey12 : Bool;   // DT12
      directKey13 : Bool;   // DT13
      directKey14 : Bool;   // DT14
      directKey15 : Bool;   // DT15
      directKey16 : Bool;   // DT16
      reserved2 : Byte;
      feedrateOvrA : Bool;
      feedrateOvrB : Bool;
      feedrateOvrC : Bool;
      feedrateOvrD : Bool;
      feedrateOvrE : Bool;
      reserved35 : Bool;
      reserved36 : Bool;
      reserved37 : Bool;
      spindleOvrA : Bool;
      spindleOvrB : Bool;
      spindleOvrC : Bool;
      spindleOvrD : Bool;
      spindleOvrE : Bool;
      reserved45 : Bool;
      reserved46 : Bool;
      reserved47 : Bool;
   END_STRUCT;
END_TYPE

TYPE "LBP_typeMcp310AdditionalOutput"
TITLE = MCP 310 image / Image du MCP 310
// Additional output image of MCP 310 / Image de sortie supplémentaire du MCP 310
   STRUCT
      reserved0 : Byte;
      reserved1 : Byte;
   END_STRUCT;
END_TYPE

TYPE "LBP_typeMcp310CPnInput"
TITLE = MCP 310C PN image / Image du MCP 310C PN
// Input image of MCP 310C PN / Image d'entrée du MCP 310C PN
   STRUCT
      standard { S7_SetPoint := 'True'} : "LBP_typeMcp310StandardInput";   // Input image of MCP 310 / Image d'entrée du MCP 310
      reserved8 : Byte;
      reserved9 : Byte;
      optionalKey1 : Bool;   // KT-IN1
      optionalKey2 : Bool;   // KT-IN2
      optionalKey3 : Bool;   // KT-IN3
      optionalKey4 : Bool;   // KT-IN4
      optionalKey5 : Bool;   // KT-IN5
      optionalKey6 : Bool;   // KT-IN6
      optionalKey7 : Bool;   // KT-IN7
      optionalKey8 : Bool;   // KT-IN8
      optionalKey9 : Bool;   // KT-IN9
      reserved111 : Bool;
      reserved112 : Bool;
      reserved113 : Bool;
      reserved114 : Bool;
      reserved115 : Bool;
      reserved116 : Bool;
      reserved117 : Bool;
      reserved12 : Byte;
      spindleOvrA : Bool;
      spindleOvrB : Bool;
      spindleOvrC : Bool;
      spindleOvrD : Bool;
      spindleOvrE : Bool;
      reserved135 : Bool;
      reserved136 : Bool;
      reserved137 : Bool;
   END_STRUCT;
END_TYPE

TYPE "LBP_typeMcp310CPnOutput"
TITLE = MCP 310C PN image / Image du MCP 310C PN
// Output image of MCP 310C PN / Image de sortie du MCP 310C PN
   STRUCT
      standard { S7_SetPoint := 'True'} : "LBP_typeMcp310StandardOutput";   // Output image of MCP 310 / Image de sortie du MCP 310
   END_STRUCT;
END_TYPE

TYPE "LBP_typeMcp310PnInput"
TITLE = MCP 310 PN image / Image du MCP 310 PN
// Input image of MCP 310 PN / Image d'entrée du MCP 310 PN
   STRUCT
      standard { S7_SetPoint := 'True'} : "LBP_typeMcp310StandardInput";   // Input image of MCP 310 / Image d'entrée du MCP 310
      directKey1 : Bool;   // DT1
      directKey2 : Bool;   // DT2
      directKey3 : Bool;   // DT3
      directKey4 : Bool;   // DT4
      directKey5 : Bool;   // DT5
      directKey6 : Bool;   // DT6
      directKey7 : Bool;   // DT7
      directKey8 : Bool;   // DT8
      directKey9 : Bool;   // DT9
      directKey10 : Bool;   // DT10
      directKey11 : Bool;   // DT11
      directKey12 : Bool;   // DT12
      directKey13 : Bool;   // DT13
      directKey14 : Bool;   // DT14
      directKey15 : Bool;   // DT15
      directKey16 : Bool;   // DT16
      optionalKey1 : Bool;   // KT-IN1
      optionalKey2 : Bool;   // KT-IN2
      optionalKey3 : Bool;   // KT-IN3
      optionalKey4 : Bool;   // KT-IN4
      optionalKey5 : Bool;   // KT-IN5
      optionalKey6 : Bool;   // KT-IN6
      optionalKey7 : Bool;   // KT-IN7
      optionalKey8 : Bool;   // KT-IN8
      optionalKey9 : Bool;   // KT-IN9
      reserved111 : Bool;
      reserved112 : Bool;
      reserved113 : Bool;
      reserved114 : Bool;
      reserved115 : Bool;
      reserved116 : Bool;
      reserved117 : Bool;
      reserved12 : Byte;
      spindleOvrA : Bool;
      spindleOvrB : Bool;
      spindleOvrC : Bool;
      spindleOvrD : Bool;
      spindleOvrE : Bool;
      reserved135 : Bool;
      reserved136 : Bool;
      reserved137 : Bool;
   END_STRUCT;
END_TYPE

TYPE "LBP_typeMcp310PnOutput"
TITLE = MCP 310 PN image / Image du MCP 310 PN
// Output image of MCP 310 PN / Image de sortie du MCP 310 PN
   STRUCT
      standard { S7_SetPoint := 'True'} : "LBP_typeMcp310StandardOutput";   // Output image of MCP 310 / Image de sortie du MCP 310
   END_STRUCT;
END_TYPE

TYPE "LBP_typeMcp310StandardInput"
TITLE = MCP 310 image / Image du MCP 310
// Input image of MCP 310 / Image d'entrée du MCP 310
   STRUCT
      auto : Bool;
      mda : Bool;
      jog : Bool;
      singleBlock : Bool;
      spindleIncrease : Bool;
      spindle100 : Bool;
      spindleDecrease : Bool;
      cycleStop : Bool;
      teachIn : Bool;
      repos : Bool;
      refPoint : Bool;
      keySwitch3 : Bool;
      spindleLeft : Bool;
      spindleStop : Bool;
      spindleRight : Bool;
      cycleStart : Bool;
      inc1 : Bool;
      inc10 : Bool;
      inc100 : Bool;
      inc1000 : Bool;
      keySwitch0 : Bool;
      incVar : Bool;
      feedrateStop : Bool;
      feedrateStart : Bool;
      feedrateOvrA : Bool;
      feedrateOvrB : Bool;
      feedrateOvrC : Bool;
      feedrateOvrD : Bool;
      feedrateOvrE : Bool;
      keySwitch1 : Bool;
      keySwitch2 : Bool;
      reset : Bool;
      optionalKey1 : Bool;   // KT-IN1
      optionalKey2 : Bool;   // KT-IN2
      optionalKey3 : Bool;   // KT-IN3
      optionalKey4 : Bool;   // KT-IN4
      optionalKey5 : Bool;   // KT-IN5
      rapidTraverse : Bool;
      minus : Bool;
      plus : Bool;
      axisX : Bool;
      axisY : Bool;
      axisZ : Bool;
      axis4 : Bool;
      axis5 : Bool;
      axis6 : Bool;
      optionalKey6 : Bool;   // KT-IN6
      customerKey16 : Bool;   // T16
      customerKey15 : Bool;   // T15
      customerKey14 : Bool;   // T14
      customerKey13 : Bool;   // T13
      mcsWcs : Bool;
      customerKey12 : Bool;   // T12
      customerKey11 : Bool;   // T11
      customerKey10 : Bool;   // T10
      customerKey9 : Bool;   // T9
      customerKey8 : Bool;   // T8
      customerKey7 : Bool;   // T7
      customerKey6 : Bool;   // T6
      customerKey5 : Bool;   // T5
      customerKey4 : Bool;   // T4
      customerKey3 : Bool;   // T3
      customerKey2 : Bool;   // T2
      customerKey1 : Bool;   // T1
   END_STRUCT;
END_TYPE

TYPE "LBP_typeMcp310StandardOutput"
TITLE = MCP 310 image / Image du MCP 310
// Output image of MCP 310 / Image de sortie du MCP 310
   STRUCT
      auto : Bool;
      mda : Bool;
      jog : Bool;
      singleBlock : Bool;
      spindleIncrease : Bool;
      spindle100 : Bool;
      spindleDecrease : Bool;
      cycleStop : Bool;
      teachIn : Bool;
      repos : Bool;
      refPoint : Bool;
      reset : Bool;
      spindleLeft : Bool;
      spindleStop : Bool;
      spindleRight : Bool;
      cycleStart : Bool;
      inc1 : Bool;
      inc10 : Bool;
      inc100 : Bool;
      inc1000 : Bool;
      reserved24 : Bool;
      incVar : Bool;
      feedrateStop : Bool;
      feedrateStart : Bool;
      reserved3 : Byte;
      optionalKey1 : Bool;   // KT-OUT1
      optionalKey2 : Bool;   // KT-OUT2
      optionalKey3 : Bool;   // KT-OUT3
      optionalKey4 : Bool;   // KT-OUT4
      optionalKey5 : Bool;   // KT-OUT5
      rapidTraverse : Bool;
      minus : Bool;
      plus : Bool;
      axisX : Bool;
      axisY : Bool;
      axisZ : Bool;
      axis4 : Bool;
      axis5 : Bool;
      axis6 : Bool;
      optionalKey6 : Bool;   // KT-OUT6
      customerKey16 : Bool;   // T16
      customerKey15 : Bool;   // T15
      customerKey14 : Bool;   // T14
      customerKey13 : Bool;   // T13
      mcsWcs : Bool;
      customerKey12 : Bool;   // T12
      customerKey11 : Bool;   // T11
      customerKey10 : Bool;   // T10
      customerKey9 : Bool;   // T9
      customerKey8 : Bool;   // T8
      customerKey7 : Bool;   // T7
      customerKey6 : Bool;   // T6
      customerKey5 : Bool;   // T5
      customerKey4 : Bool;   // T4
      customerKey3 : Bool;   // T3
      customerKey2 : Bool;   // T2
      customerKey1 : Bool;   // T1
   END_STRUCT;
END_TYPE

TYPE "LBP_typeMcp483AdditionalInput"
TITLE = MCP 483 image / Image du MCP 483
// Additional input image of MCP 483 / Image d'entrée supplémentaire du MCP 483
   STRUCT
      directKey1 : Bool;   // DT1
      directKey2 : Bool;   // DT2
      directKey3 : Bool;   // DT3
      directKey4 : Bool;   // DT4
      directKey5 : Bool;   // DT5
      directKey6 : Bool;   // DT6
      directKey7 : Bool;   // DT7
      directKey8 : Bool;   // DT8
      directKey9 : Bool;   // DT9
      directKey10 : Bool;   // DT10
      directKey11 : Bool;   // DT11
      directKey12 : Bool;   // DT12
      directKey13 : Bool;   // DT13
      directKey14 : Bool;   // DT14
      directKey15 : Bool;   // DT15
      directKey16 : Bool;   // DT16
      optionalKey1 : Bool;   // KT-IN1
      optionalKey2 : Bool;   // KT-IN2
      optionalKey3 : Bool;   // KT-IN3
      optionalKey4 : Bool;   // KT-IN4
      optionalKey5 : Bool;   // KT-IN5
      optionalKey6 : Bool;   // KT-IN6
      reserved26 : Bool;
      reserved27 : Bool;
      feedrateOvrA : Bool;
      feedrateOvrB : Bool;
      feedrateOvrC : Bool;
      feedrateOvrD : Bool;
      feedrateOvrE : Bool;
      reserved35 : Bool;
      reserved36 : Bool;
      reserved37 : Bool;
      spindleOvrA : Bool;
      spindleOvrB : Bool;
      spindleOvrC : Bool;
      spindleOvrD : Bool;
      spindleOvrE : Bool;
      reserved45 : Bool;
      reserved46 : Bool;
      reserved47 : Bool;
   END_STRUCT;
END_TYPE

TYPE "LBP_typeMcp483AdditionalOutput"
TITLE = MCP 483 image / Image du MCP 483
// Additional output image of MCP 483 / Image de sortie supplémentaire du MCP 483
   STRUCT
      reserved1 : Byte;
      optionalKey1 : Bool;   // KT-OUT1,
      optionalKey2 : Bool;   // KT-OUT2
      optionalKey3 : Bool;   // KT-OUT3
      optionalKey4 : Bool;   // KT-OUT4
      optionalKey5 : Bool;   // KT-OUT5
      optionalKey6 : Bool;   // KT-OUT6
      reserved16 : Bool;
      reserved17 : Bool;
   END_STRUCT;
END_TYPE

TYPE "LBP_typeMcp483CPnInput"
TITLE = MCP 483C PN image / Image du MCP 483C PN
// Input image of MCP 483C PN / Image d'entrée du MCP 483C PN
   STRUCT
      standard { S7_SetPoint := 'True'} : "LBP_typeMcp483StandardInput";   // Input image of MCP 483 / Image d'entrée du MCP 483
      reserved8 : Byte;
      reserved9 : Byte;
      optionalKey1 : Bool;   // KT-IN1
      optionalKey2 : Bool;   // KT-IN2
      optionalKey3 : Bool;   // KT-IN3
      optionalKey4 : Bool;   // KT-IN4
      optionalKey5 : Bool;   // KT-IN5
      optionalKey6 : Bool;   // KT-IN6
      optionalKey7 : Bool;   // KT-IN7
      optionalKey8 : Bool;   // KT-IN8
      optionalKey9 : Bool;   // KT-IN9
      reserved111 : Bool;
      reserved112 : Bool;
      reserved113 : Bool;
      reserved114 : Bool;
      reserved115 : Bool;
      reserved116 : Bool;
      reserved117 : Bool;
      reserved12 : Byte;
      spindleOvrA : Bool;
      spindleOvrB : Bool;
      spindleOvrC : Bool;
      spindleOvrD : Bool;
      spindleOvrE : Bool;
      reserved135 : Bool;
      reserved136 : Bool;
      reserved137 : Bool;
   END_STRUCT;
END_TYPE

TYPE "LBP_typeMcp483CPnOutput"
TITLE = MCP 483C PN image / Image du MCP 483C PN
// Output image of MCP 483C PN / Image de sortie du MCP 483C PN
   STRUCT
      standard { S7_SetPoint := 'True'} : "LBP_typeMcp483StandardOutput";   // Output image of MCP 483 / Image de sortie du MCP 483
   END_STRUCT;
END_TYPE

TYPE "LBP_typeMcp483MillingInput"
TITLE = MCP 483 image / Image du MCP 483
// Input image of MCP 483 Milling / Image d'entrée du MCP 483 Fraisage
   STRUCT
      auto : Bool;
      mda : Bool;
      teachIn : Bool;
      jog : Bool;
      spindleOvrA : Bool;
      spindleOvrB : Bool;
      spindleOvrC : Bool;
      spindleOvrD : Bool;
      inc1 : Bool;
      inc10 : Bool;
      inc100 : Bool;
      inc1000 : Bool;
      inc10000 : Bool;
      incVar : Bool;
      refPoint : Bool;
      repos : Bool;
      cycleStop : Bool;
      cycleStart : Bool;
      feedrateStop : Bool;
      feedrateStart : Bool;
      spindleStop : Bool;
      spindleStart : Bool;
      keySwitch2 : Bool;
      keySwitch0 : Bool;
      feedrateOvrA : Bool;
      feedrateOvrB : Bool;
      feedrateOvrC : Bool;
      feedrateOvrD : Bool;
      feedrateOvrE : Bool;
      singleBlock : Bool;
      keySwitch1 : Bool;
      reset : Bool;
      axis10 : Bool;   // R10
      axis7 : Bool;   // R7
      axis4 : Bool;   // R4
      axisX : Bool;   // R1
      keySwitch3 : Bool;
      rapidTraverse : Bool;   // R14
      minus : Bool;   // R13
      plus : Bool;   // R15
      axis6 : Bool;   // R6
      axis8 : Bool;   // R8
      axis9 : Bool;   // R9
      tcs : Bool;   // R11
      mcsWcs : Bool;   // R12
      axis5 : Bool;   // R5
      axisZ : Bool;   // R3
      axisY : Bool;   // R2
      reserved60 : Bool;
      customerKey15 : Bool;   // T15
      customerKey14 : Bool;   // T14
      customerKey13 : Bool;   // T13
      customerKey12 : Bool;   // T12
      customerKey11 : Bool;   // T11
      customerKey10 : Bool;   // T10
      customerKey9 : Bool;   // T9
      customerKey8 : Bool;   // T8
      customerKey7 : Bool;   // T7
      customerKey6 : Bool;   // T6
      customerKey5 : Bool;   // T5
      customerKey4 : Bool;   // T4
      customerKey3 : Bool;   // T3
      customerKey2 : Bool;   // T2
      customerKey1 : Bool;   // T1
   END_STRUCT;
END_TYPE

TYPE "LBP_typeMcp483MillingOutput"
TITLE = MCP 483 image / Image du MCP 483
// Output image of MCP 483 Milling / Image de sortie du MCP 483 Fraisage
   STRUCT
      auto : Bool;
      mda : Bool;
      teachIn : Bool;
      jog : Bool;
      inc1 : Bool;
      inc10 : Bool;
      inc100 : Bool;
      inc1000 : Bool;
      inc10000 : Bool;
      incVar : Bool;
      refPoint : Bool;
      repos : Bool;
      cycleStop : Bool;
      cycleStart : Bool;
      feedrateStop : Bool;
      feedrateStart : Bool;
      spindleStop : Bool;
      spindleStart : Bool;
      singleBlock : Bool;
      axis10 : Bool;   // R10
      axis7 : Bool;   // R7
      axis4 : Bool;   // R4
      axisX : Bool;   // R1
      minus : Bool;   // R13
      plus : Bool;   // R15
      axis6 : Bool;   // R6
      axis8 : Bool;   // R8
      axis9 : Bool;   // R9
      tcs : Bool;   // R11
      mcsWcs : Bool;   // R12
      axis5 : Bool;   // R5
      axisZ : Bool;   // R3
      axisY : Bool;   // R2
      customerKey15 : Bool;   // T15
      customerKey14 : Bool;   // T14
      customerKey13 : Bool;   // T13
      customerKey12 : Bool;   // T12
      customerKey11 : Bool;   // T11
      customerKey10 : Bool;   // T10
      customerKey9 : Bool;   // T9
      customerKey8 : Bool;   // T8
      customerKey7 : Bool;   // T7
      customerKey6 : Bool;   // T6
      customerKey5 : Bool;   // T5
      customerKey4 : Bool;   // T4
      customerKey3 : Bool;   // T3
      customerKey2 : Bool;   // T2
      customerKey1 : Bool;   // T1
   END_STRUCT;
END_TYPE

TYPE "LBP_typeMcp483PnInput"
TITLE = MCP 483 PN image / Image du MCP 483 PN
// Input image of MCP 483 PN / Image d'entrée du MCP 483 PN
   STRUCT
      standard { S7_SetPoint := 'True'} : "LBP_typeMcp483StandardInput";   // Input image of MCP 483 / Image d'entrée du MCP 483
      directKey1 : Bool;   // DT1
      directKey2 : Bool;   // DT2
      directKey3 : Bool;   // DT3
      directKey4 : Bool;   // DT4
      directKey5 : Bool;   // DT5
      directKey6 : Bool;   // DT6
      directKey7 : Bool;   // DT7
      directKey8 : Bool;   // DT8
      directKey9 : Bool;   // DT9
      directKey10 : Bool;   // DT10
      directKey11 : Bool;   // DT11
      directKey12 : Bool;   // DT12
      directKey13 : Bool;   // DT13
      directKey14 : Bool;   // DT14
      directKey15 : Bool;   // DT15
      directKey16 : Bool;   // DT16
      optionalKey1 : Bool;   // KT-IN1
      optionalKey2 : Bool;   // KT-IN2
      optionalKey3 : Bool;   // KT-IN3
      optionalKey4 : Bool;   // KT-IN4
      optionalKey5 : Bool;   // KT-IN5
      optionalKey6 : Bool;   // KT-IN6
      optionalKey7 : Bool;   // KT-IN7
      optionalKey8 : Bool;   // KT-IN8
      optionalKey9 : Bool;   // KT-IN9
      reserved111 : Bool;
      reserved112 : Bool;
      reserved113 : Bool;
      reserved114 : Bool;
      reserved115 : Bool;
      reserved116 : Bool;
      reserved117 : Bool;
      reserved12 : Byte;
      spindleOvrA : Bool;
      spindleOvrB : Bool;
      spindleOvrC : Bool;
      spindleOvrD : Bool;
      spindleOvrE : Bool;
      reserved135 : Bool;
      reserved136 : Bool;
      reserved137 : Bool;
   END_STRUCT;
END_TYPE

TYPE "LBP_typeMcp483PnOutput"
TITLE = MCP 483 PN image / Image du MCP 483 PN
// Output image of MCP 483 PN / Image de sortie du MCP 483 PN
   STRUCT
      standard { S7_SetPoint := 'True'} : "LBP_typeMcp483StandardOutput";   // Output image of MCP 483 / Image de sortie du MCP 483
   END_STRUCT;
END_TYPE

TYPE "LBP_typeMcp483StandardInput"
TITLE = MCP 483 image / Image du MCP 483
// Input image of MCP 483 / Image d'entrée du MCP 483
   STRUCT
      auto : Bool;
      mda : Bool;
      teachIn : Bool;
      jog : Bool;
      spindleOvrA : Bool;
      spindleOvrB : Bool;
      spindleOvrC : Bool;
      spindleOvrD : Bool;
      inc1 : Bool;
      inc10 : Bool;
      inc100 : Bool;
      inc1000 : Bool;
      inc10000 : Bool;
      incVar : Bool;
      refPoint : Bool;
      repos : Bool;
      cycleStop : Bool;
      cycleStart : Bool;
      feedrateStop : Bool;
      feedrateStart : Bool;
      spindleStop : Bool;
      spindleStart : Bool;
      keySwitch2 : Bool;
      keySwitch0 : Bool;
      feedrateOvrA : Bool;
      feedrateOvrB : Bool;
      feedrateOvrC : Bool;
      feedrateOvrD : Bool;
      feedrateOvrE : Bool;
      singleBlock : Bool;
      keySwitch1 : Bool;
      reset : Bool;
      axis10 : Bool;   // R10
      axis7 : Bool;   // R7
      axis4 : Bool;   // R4
      axisX : Bool;   // R1
      keySwitch3 : Bool;
      rapidTraverse : Bool;   // R14
      minus : Bool;   // R13
      plus : Bool;   // R15
      axis6 : Bool;   // R6
      axis8 : Bool;   // R8
      axis9 : Bool;   // R9
      axis11 : Bool;   // R11
      mcsWcs : Bool;   // R12
      axis5 : Bool;   // R5
      axisZ : Bool;   // R3
      axisY : Bool;   // R2
      reserved60 : Bool;
      customerKey15 : Bool;   // T15
      customerKey14 : Bool;   // T14
      customerKey13 : Bool;   // T13
      customerKey12 : Bool;   // T12
      customerKey11 : Bool;   // T11
      customerKey10 : Bool;   // T10
      customerKey9 : Bool;   // T9
      customerKey8 : Bool;   // T8
      customerKey7 : Bool;   // T7
      customerKey6 : Bool;   // T6
      customerKey5 : Bool;   // T5
      customerKey4 : Bool;   // T4
      customerKey3 : Bool;   // T3
      customerKey2 : Bool;   // T2
      customerKey1 : Bool;   // T1
   END_STRUCT;
END_TYPE

TYPE "LBP_typeMcp483StandardOutput"
TITLE = MCP 483 image / Image du MCP 483
// Output image of MCP 483 / Image de sortie du MCP 483
   STRUCT
      LEDauto : Bool;
      LEDmda : Bool;
      LEDteachIn : Bool;
      LEDjog : Bool;
      LEDinc1 : Bool;
      LEDinc10 : Bool;
      LEDinc100 : Bool;
      LEDinc1000 : Bool;
      LEDinc10000 : Bool;
      LEDincVar : Bool;
      LEDrefPoint : Bool;
      LEDrepos : Bool;
      LEDcycleStop : Bool;
      LEDcycleStart : Bool;
      LEDfeedrateStop : Bool;
      LEDfeedrateStart : Bool;
      LEDspindleStop : Bool;
      LEDspindleStart : Bool;
      LEDsingleBlock : Bool;
      LEDaxis10 : Bool;   // R10
      LEDaxis7 : Bool;   // R7
      LEDaxis4 : Bool;   // R4
      LEDaxisX : Bool;   // R1
      LEDminus : Bool;   // R13
      LEDplus : Bool;   // R15
      LEDaxis6 : Bool;   // R6
      LEDaxis8 : Bool;   // R8
      LEDaxis9 : Bool;   // R9
      LEDaxis11 : Bool;   // R11
      LEDmcsWcs : Bool;   // R12
      LEDaxis5 : Bool;   // R5
      LEDaxisZ : Bool;   // R3
      LEDaxisY : Bool;   // R2
      LEDcustomerKey15 : Bool;   // T15
      LEDcustomerKey14 : Bool;   // T14
      LEDcustomerKey13 : Bool;   // T13
      LEDcustomerKey12 : Bool;   // T12
      LEDcustomerKey11 : Bool;   // T11
      LEDcustomerKey10 : Bool;   // T10
      LEDcustomerKey9 : Bool;   // T9
      LEDcustomerKey8 : Bool;   // T8
      LEDcustomerKey7 : Bool;   // T7
      LEDcustomerKey6 : Bool;   // T6
      LEDcustomerKey5 : Bool;   // T5
      LEDcustomerKey4 : Bool;   // T4
      LEDcustomerKey3 : Bool;   // T3
      LEDcustomerKey2 : Bool;   // T2
      LEDcustomerKey1 : Bool;   // T1
      LEDrapidTraverse : Bool;   // R14
      LEDreset : Bool;
      reserved62 : Bool;
      reserved63 : Bool;
      reserved64 : Bool;
      reserved65 : Bool;
      reserved66 : Bool;
      reserved67 : Bool;
      LEDoptionalKey1 : Bool;   // KT-OUT1, reserved / KT-OUT1, réservé
      LEDoptionalKey2 : Bool;   // KT-OUT2, reserved / KT-OUT2, réservé
      LEDoptionalKey3 : Bool;   // KT-OUT3, reserved / KT-OUT3, réservé
      LEDoptionalKey4 : Bool;   // KT-OUT4, reserved / KT-OUT4, réservé
      LEDoptionalKey5 : Bool;   // KT-OUT5, reserved / KT-OUT5, réservé
      LEDoptionalKey6 : Bool;   // KT-OUT6, reserved / KT-OUT6, réservé
      reserved76 : Bool;
      reserved77 : Bool;
   END_STRUCT;
END_TYPE

TYPE "LBP_typeMcp483TurningInput"
TITLE = MCP 483 image / Image du MCP 483
// Input image of MCP 483 Turning / Image d'entrée du MCP 483 Tournage
   STRUCT
      auto : Bool;
      mda : Bool;
      teachIn : Bool;
      jog : Bool;
      spindleOvrA : Bool;
      spindleOvrB : Bool;
      spindleOvrC : Bool;
      spindleOvrD : Bool;
      inc1 : Bool;
      inc10 : Bool;
      inc100 : Bool;
      inc1000 : Bool;
      inc10000 : Bool;
      incVar : Bool;
      refPoint : Bool;
      repos : Bool;
      cycleStop : Bool;
      cycleStart : Bool;
      feedrateStop : Bool;
      feedrateStart : Bool;
      spindleStop : Bool;
      spindleStart : Bool;
      keySwitch2 : Bool;
      keySwitch0 : Bool;
      feedrateOvrA : Bool;
      feedrateOvrB : Bool;
      feedrateOvrC : Bool;
      feedrateOvrD : Bool;
      feedrateOvrE : Bool;
      singleBlock : Bool;
      keySwitch1 : Bool;
      reset : Bool;
      r10 : Bool;   // R10
      axisCMinus : Bool;   // R7
      axisZMinus : Bool;   // R4
      axisYPlus : Bool;   // R1
      keySwitch3 : Bool;
      r14 : Bool;   // R14
      r13 : Bool;   // R13
      r15 : Bool;   // R15
      axisZPlus : Bool;   // R6
      axisXMinus : Bool;   // R8
      axisYMinus : Bool;   // R9
      r11 : Bool;   // R11
      mcsWcs : Bool;   // R12
      rapidTraverse : Bool;   // R5
      axisCPlus : Bool;   // R3
      axisXPlus : Bool;   // R2
      reserved60 : Bool;
      customerKey15 : Bool;   // T15
      customerKey14 : Bool;   // T14
      customerKey13 : Bool;   // T13
      customerKey12 : Bool;   // T12
      customerKey11 : Bool;   // T11
      customerKey10 : Bool;   // T10
      customerKey9 : Bool;   // T9
      customerKey8 : Bool;   // T8
      customerKey7 : Bool;   // T7
      customerKey6 : Bool;   // T6
      customerKey5 : Bool;   // T5
      customerKey4 : Bool;   // T4
      customerKey3 : Bool;   // T3
      customerKey2 : Bool;   // T2
      customerKey1 : Bool;   // T1
   END_STRUCT;
END_TYPE

TYPE "LBP_typeMcp483TurningOutput"
TITLE = MCP 483 image / Image du MCP 483
// Output image of MCP 483 Turning / Image de sortie du MCP 483 Tournage
   STRUCT
      auto : Bool;
      mda : Bool;
      teachIn : Bool;
      jog : Bool;
      inc1 : Bool;
      inc10 : Bool;
      inc100 : Bool;
      inc1000 : Bool;
      inc10000 : Bool;
      incVar : Bool;
      refPoint : Bool;
      repos : Bool;
      cycleStop : Bool;
      cycleStart : Bool;
      feedrateStop : Bool;
      feedrateStart : Bool;
      spindleStop : Bool;
      spindleStart : Bool;
      singleBlock : Bool;
      r10 : Bool;   // R10
      axisCMinus : Bool;   // R7
      axisZMinus : Bool;   // R4
      axisYPlus : Bool;   // R1
      r13 : Bool;   // R13
      r15 : Bool;   // R15
      axisZPlus : Bool;   // R6
      axisXMinus : Bool;   // R8
      axisYMinus : Bool;   // R9
      r11 : Bool;   // R11
      mcsWcs : Bool;   // R12
      rapidTraverse : Bool;   // R5
      axisCPlus : Bool;   // R3
      axisXPlus : Bool;   // R2
      customerKey15 : Bool;   // T15
      customerKey14 : Bool;   // T14
      customerKey13 : Bool;   // T13
      customerKey12 : Bool;   // T12
      customerKey11 : Bool;   // T11
      customerKey10 : Bool;   // T10
      customerKey9 : Bool;   // T9
      customerKey8 : Bool;   // T8
      customerKey7 : Bool;   // T7
      customerKey6 : Bool;   // T6
      customerKey5 : Bool;   // T5
      customerKey4 : Bool;   // T4
      customerKey3 : Bool;   // T3
      customerKey2 : Bool;   // T2
      customerKey1 : Bool;   // T1
   END_STRUCT;
END_TYPE

TYPE "LBP_typeModularMcpAxisInput"
TITLE = Modular MCP image / Image MCP modulaire
// Input image of axis keypad for modular MCP / Image des entrées du champ de touches d'axe pour MCP modulaires
   STRUCT
      minus : Bool;   // input image n+0 bit 0 / Image des entrées n+0 bit 0
      rapidTraverse : Bool;   // input image n+0 bit 1 / Image des entrées n+0 bit 1
      plus : Bool;   // input image n+0 bit 2 / Image des entrées n+0 bit 2
      key3 : Bool;   // input image n+0 bit 3 / Image des entrées n+0 bit 3
      tcs : Bool;   // input image n+0 bit 4 / Image des entrées n+0 bit 4
      mcsWcs : Bool;   // input image n+0 bit 5 / Image des entrées n+0 bit 5
      key6 : Bool;   // input image n+0 bit 6 / Image des entrées n+0 bit 6
      key7 : Bool;   // input image n+0 bit 7 / Image des entrées n+0 bit 7
      key8 : Bool;   // input image n+1 bit 0 / Image des entrées n+1 bit 0
      axis4 : Bool;   // input image n+1 bit 1 / Image des entrées n+1 bit 1
      axis5 : Bool;   // input image n+1 bit 2 / Image des entrées n+1 bit 2
      axis6 : Bool;   // input image n+1 bit 3 / Image des entrées n+1 bit 3
      axisX : Bool;   // input image n+1 bit 4 / Image des entrées n+1 bit 4
      axisY : Bool;   // input image n+1 bit 5 / Image des entrées n+1 bit 5
      axisZ : Bool;   // input image n+1 bit 6 / Image des entrées n+1 bit 6
      reserved17 : Bool;
      feedrateStop : Bool;   // input image n+2 bit 0 / Image des entrées n+2 bit 0
      feedrateStart : Bool;   // input image n+2 bit 1 / Image des entrées n+2 bit 1
      key18 : Bool;   // input image n+2 bit 2 / Image des entrées n+2 bit 2
      reserved23 : Bool;
      reserved24 : Bool;
      reserved25 : Bool;
      reserved26 : Bool;
      reserved27 : Bool;
      spindleStop : Bool;   // input image n+3 bit 0 / Image des entrées n+3 bit 0
      spindleStart : Bool;   // input image n+3 bit 1 / Image des entrées n+3 bit 1
      key26 : Bool;   // input image n+3 bit 2 / Image des entrées n+3 bit 2
      reserved33 : Bool;
      reserved34 : Bool;
      reserved35 : Bool;
      reserved36 : Bool;
      reserved37 : Bool;
   END_STRUCT;
END_TYPE

TYPE "LBP_typeModularMcpAxisOutput"
TITLE = Modular MCP image / Image MCP modulaire
// Output image of axis keypad for modular MCP / Image des sorties du champ de touches d'axe pour MCP modulaires
   STRUCT
      minus : Bool;   // output image n+0 bit 0 / Image des sorties n+0 bit 0
      rapidTraverse : Bool;   // output image n+0 bit 1 / Image des sorties n+0 bit 1
      plus : Bool;   // output image n+0 bit 2 / Image des sorties n+0 bit 2
      led3 : Bool;   // output image n+0 bit 3 / Image des sorties n+0 bit 3
      tcs : Bool;   // output image n+0 bit 4 / Image des sorties n+0 bit 4
      mcsWcs : Bool;   // output image n+0 bit 5 / Image des sorties n+0 bit 5
      led6 : Bool;   // output image n+0 bit 6 / Image des sorties n+0 bit 6
      led7 : Bool;   // output image n+0 bit 7 / Image des sorties n+0 bit 7
      led8 : Bool;   // output image n+1 bit 0 / Image des sorties n+1 bit 0
      axis4 : Bool;   // output image n+1 bit 1 / Image des sorties n+1 bit 1
      axis5 : Bool;   // output image n+1 bit 2 / Image des sorties n+1 bit 2
      axis6 : Bool;   // output image n+1 bit 3 / Image des sorties n+1 bit 3
      axisX : Bool;   // output image n+1 bit 4 / Image des sorties n+1 bit 4
      axisY : Bool;   // output image n+1 bit 5 / Image des sorties n+1 bit 5
      axisZ : Bool;   // output image n+1 bit 6 / Image des sorties n+1 bit 6
      reserved17 : Bool;
      feedrateStop : Bool;   // output image n+2 bit 0 / Image des sorties n+2 bit 0
      feedrateStart : Bool;   // output image n+2 bit 1 / Image des sorties n+2 bit 1
      led18 : Bool;   // output image n+2 bit 2 / Image des sorties n+2 bit 2
      reserved23 : Bool;
      reserved24 : Bool;
      reserved25 : Bool;
      reserved26 : Bool;
      reserved27 : Bool;
      spindleStop : Bool;   // output image n+3 bit 0 / Image des sorties n+3 bit 0
      spindleStart : Bool;   // output image n+3 bit 1 / Image des sorties n+3 bit 1
      led26 : Bool;   // output image n+3 bit 2 / Image des sorties n+3 bit 2
      reserved33 : Bool;
      reserved34 : Bool;
      reserved35 : Bool;
      reserved36 : Bool;
      reserved37 : Bool;
   END_STRUCT;
END_TYPE

TYPE "LBP_typeModularMcpBaseInput"
TITLE = Modular MCP image / Image MCP modulaire
// Input image of base signals for modular MCP / Image des entrées des signaux de base pour MCP modulaires
   STRUCT
      optionalKey1 : Bool;   // input image n+0 bit 0; KT-IN1 / Image des entrées n+0 bit 0 ; KT-IN1
      optionalKey2 : Bool;   // input image n+0 bit 1; KT-IN2 / Image des entrées n+0 bit 1 ; KT-IN2
      optionalKey3 : Bool;   // input image n+0 bit 2; KT-IN3 / Image des entrées n+0 bit 2 ; KT-IN3
      optionalKey4 : Bool;   // input image n+0 bit 3; KT-IN4 / Image des entrées n+0 bit 3 ; KT-IN4
      optionalKey5 : Bool;   // input image n+0 bit 4; KT-IN5 / Image des entrées n+0 bit 4 ; KT-IN5
      optionalKey6 : Bool;   // input image n+0 bit 5; KT-IN6 / Image des entrées n+0 bit 5 ; KT-IN6
      optionalKey7 : Bool;   // input image n+0 bit 6; KT-IN7 / Image des entrées n+0 bit 6 ; KT-IN7
      optionalKey8 : Bool;   // input image n+0 bit 7; KT-IN8 / Image des entrées n+0 bit 7 ; KT-IN8
      optionalKey9 : Bool;   // input image n+1 bit 0; KT-IN9 / Image des entrées n+1 bit 0 ; KT-IN9
      optionalKey10 : Bool;   // input image n+1 bit 1; KT-IN10 / Image des entrées n+1 bit 1 ; KT-IN10
      optionalKey11 : Bool;   // input image n+1 bit 2; KT-IN11 / Image des entrées n+1 bit 2 ; KT-IN11
      optionalKey12 : Bool;   // input image n+1 bit 3; KT-IN12 / Image des entrées n+1 bit 3 ; KT-IN12
      optionalKey13 : Bool;   // input image n+1 bit 4; KT-IN13 / Image des entrées n+1 bit 4 ; KT-IN13
      optionalKey14 : Bool;   // input image n+1 bit 5; KT-IN14 / Image des entrées n+1 bit 5 ; KT-IN14
      optionalKey15 : Bool;   // input image n+1 bit 6; KT-IN15 / Image des entrées n+1 bit 6 ; KT-IN15
      optionalKey16 : Bool;   // input image n+1 bit 7; KT-IN16 / Image des entrées n+1 bit 7 ; KT-IN16
      spindleOvr : USInt;   // input image byte n+2 / Image des entrées octet n+2
      feedrateOvr : USInt;   // input image byte n+3 / Image des entrées octet n+3
      keySwitch0 : Bool;   // input image n+4 bit 0 / Image des entrées n+4 bit 0
      keySwitch1 : Bool;   // input image n+4 bit 1 / Image des entrées n+4 bit 1
      keySwitch2 : Bool;   // input image n+4 bit 2 / Image des entrées n+4 bit 2
      keySwitch3 : Bool;   // input image n+4 bit 3 / Image des entrées n+4 bit 3
      reserved44 : Bool;
      reserved45 : Bool;
      reserved46 : Bool;
      reserved47 : Bool;
      reserved50 : Bool;
      reserved51 : Bool;
      reserved52 : Bool;
      reserved53 : Bool;
      reserved54 : Bool;
      reserved55 : Bool;
      reserved56 : Bool;
      reserved57 : Bool;
   END_STRUCT;
END_TYPE

TYPE "LBP_typeModularMcpBaseOutput"
TITLE = Modular MCP image / Image MCP modulaire
// Output image of base signals for modular MCP / Image des sorties des signaux de base pour MCP modulaires
   STRUCT
      optionalKey1 : Bool;   // output image n+0 bit 0; KT-OUT1 / Image des sorties n+0 bit 0 ; KT-OUT1
      optionalKey2 : Bool;   // output image n+0 bit 1; KT-OUT2 / Image des sorties n+0 bit 1 ; KT-OUT2
      optionalKey3 : Bool;   // output image n+0 bit 2; KT-OUT3 / Image des sorties n+0 bit 2 ; KT-OUT3
      optionalKey4 : Bool;   // output image n+0 bit 3; KT-OUT4 / Image des sorties n+0 bit 3 ; KT-OUT4
      optionalKey5 : Bool;   // output image n+0 bit 4; KT-OUT5 / Image des sorties n+0 bit 4 ; KT-OUT5
      optionalKey6 : Bool;   // output image n+0 bit 5; KT-OUT6 / Image des sorties n+0 bit 5 ; KT-OUT6
      optionalKey7 : Bool;   // output image n+0 bit 6; KT-OUT7 / Image des sorties n+0 bit 6 ; KT-OUT7
      optionalKey8 : Bool;   // output image n+0 bit 7; KT-OUT8 / Image des sorties n+0 bit 7 ; KT-OUT8
      optionalKey9 : Bool;   // output image n+1 bit 0; KT-OUT9 / Image des sorties n+1 bit 0 ; KT-OUT9
      optionalKey10 : Bool;   // output image n+1 bit 1; KT-OUT10 / Image des sorties n+1 bit 1 ; KT-OUT10
      optionalKey11 : Bool;   // output image n+1 bit 2; KT-OUT11 / Image des sorties n+1 bit 2 ; KT-OUT11
      optionalKey12 : Bool;   // output image n+1 bit 3; KT-OUT12 / Image des sorties n+1 bit 3 ; KT-OUT12
      optionalKey13 : Bool;   // output image n+1 bit 4; KT-OUT13 / Image des sorties n+1 bit 4 ; KT-OUT13
      optionalKey14 : Bool;   // output image n+1 bit 5; KT-OUT14 / Image des sorties n+1 bit 5 ; KT-OUT14
      optionalKey15 : Bool;   // output image n+1 bit 6; KT-OUT15 / Image des sorties n+1 bit 6 ; KT-OUT15
      optionalKey16 : Bool;   // output image n+1 bit 7; KT-OUT16 / Image des sorties n+1 bit 7 ; KT-OUT16
   END_STRUCT;
END_TYPE

TYPE "LBP_typeModularMcpKeypadRecord"
TITLE = Modular MCP image / Image MCP modulaire
// Image of modular MCP for key properties / Image des MCP modulaires pour propriétés des touches
   STRUCT
      recordVersion : Byte := 16#10;   // version 1.0
      keyActiveAttributesCount : USInt;   // number of valid entries in keyActiveAttributes / nombre d'entrées valides dans keyActiveAttributes
      keyInactiveAttributesCount : USInt;   // number of valid entries in keyInactiveAttributes / nombre d'entrées valides dans keyInactiveAttributes
      reserved : Byte;   // unused variable / variable inutilisée
      keyActiveAttributes { S7_SetPoint := 'True'} : Array[0..20] of "LBP_typeModularMcpLedAttribute";   // color attributes for keys in state "active" / attributs de couleur pour les touches à l'état "actif"
      keyInactiveAttributes { S7_SetPoint := 'True'} : Array[0..20] of "LBP_typeModularMcpLedAttribute";   // color attributes for keys in state "inactive" / attributs de couleur pour les touches à l'état "inactif"
   END_STRUCT;
END_TYPE

TYPE "LBP_typeModularMcpLedAttribute"
TITLE = Modular MCP image / Image MCP modulaire
// User data type for LBP_typeModularMcpKeypadRecord (sub type) / Type de données utilisateur pour LBP_typeModularMcpKeypadRecord (sous-type)
   STRUCT
      keyIndex : USInt;   // index of key / indice de touche
      red : USInt;   // intensity of red LED / intensité de la LED rouge
      green : USInt;   // intensity of green LED / intensité de la LED verte
      blue : USInt;   // intensity of blue LED / intensité de la LED bleue
   END_STRUCT;
END_TYPE

TYPE "LBP_typeModularMcpModeGroupInput"
TITLE = Modular MCP image / Image MCP modulaire
// Input image of mode group keypad for modular MCP / Image des entrées du pupitre de groupes de modes de fonctionnement pour MCP modulaires
   STRUCT
      reset : Bool;   // input image n+0 bit 0 / Image des entrées n+0 bit 0
      cycleStop : Bool;   // input image n+0 bit 1 / Image des entrées n+0 bit 1
      cycleStart : Bool;   // input image n+0 bit 2 / Image des entrées n+0 bit 2
      singleBlock : Bool;   // input image n+0 bit 3 / Image des entrées n+0 bit 3
      inc100 : Bool;   // input image n+0 bit 4 / Image des entrées n+0 bit 4
      inc1000 : Bool;   // input image n+0 bit 5 / Image des entrées n+0 bit 5
      auto : Bool;   // input image n+0 bit 6 / Image des entrées n+0 bit 6
      inc1 : Bool;   // input image n+0 bit 7 / Image des entrées n+0 bit 7
      inc10 : Bool;   // input image n+1 bit 0 / Image des entrées n+1 bit 0
      mda : Bool;   // input image n+1 bit 1 / Image des entrées n+1 bit 1
      teachIn : Bool;   // input image n+1 bit 2 / Image des entrées n+1 bit 2
      incVar : Bool;   // input image n+1 bit 3 / Image des entrées n+1 bit 3
      jog : Bool;   // input image n+1 bit 4 / Image des entrées n+1 bit 4
      repos : Bool;   // input image n+1 bit 5 / Image des entrées n+1 bit 5
      refPoint : Bool;   // input image n+1 bit 6 / Image des entrées n+1 bit 6
      reserved17 : Bool;
      key16 : Bool;   // input image n+2 bit 0 / Image des entrées n+2 bit 0
      key17 : Bool;   // input image n+2 bit 1 / Image des entrées n+2 bit 1
      key18 : Bool;   // input image n+2 bit 2 / Image des entrées n+2 bit 2
      reserved23 : Bool;
      reserved24 : Bool;
      reserved25 : Bool;
      reserved26 : Bool;
      reserved27 : Bool;
      key24 : Bool;   // input image n+3 bit 0 / Image des entrées n+3 bit 0
      key25 : Bool;   // input image n+3 bit 1 / Image des entrées n+3 bit 1
      key26 : Bool;   // input image n+3 bit 2 / Image des entrées n+3 bit 2
      reserved33 : Bool;
      reserved34 : Bool;
      reserved35 : Bool;
      reserved36 : Bool;
      reserved37 : Bool;
   END_STRUCT;
END_TYPE

TYPE "LBP_typeModularMcpModeGroupOutput"
TITLE = Modular MCP image / Image MCP modulaire
// Output image of mode group keypad for modular MCP / Image des sorties du pupitre de groupes de modes de fonctionnement pour MCP modulaires
   STRUCT
      reset : Bool;   // output image n+0 bit 0 / Image des sorties n+0 bit 0
      cycleStop : Bool;   // output image n+0 bit 1 / Image des sorties n+0 bit 1
      cycleStart : Bool;   // output image n+0 bit 2 / Image des sorties n+0 bit 2
      singleBlock : Bool;   // output image n+0 bit 3 / Image des sorties n+0 bit 3
      inc100 : Bool;   // output image n+0 bit 4 / Image des sorties n+0 bit 4
      inc1000 : Bool;   // output image n+0 bit 5 / Image des sorties n+0 bit 5
      auto : Bool;   // output image n+0 bit 6 / Image des sorties n+0 bit 6
      inc1 : Bool;   // output image n+0 bit 7 / Image des sorties n+0 bit 7
      inc10 : Bool;   // output image n+1 bit 0 / Image des sorties n+1 bit 0
      mda : Bool;   // output image n+1 bit 1 / Image des sorties n+1 bit 1
      teachIn : Bool;   // output image n+1 bit 2 / Image des sorties n+1 bit 2
      incVar : Bool;   // output image n+1 bit 3 / Image des sorties n+1 bit 3
      jog : Bool;   // output image n+1 bit 4 / Image des sorties n+1 bit 4
      repos : Bool;   // output image n+1 bit 5 / Image des sorties n+1 bit 5
      refPoint : Bool;   // output image n+1 bit 6 / Image des sorties n+1 bit 6
      reserved17 : Bool;
      led16 : Bool;   // output image n+2 bit 0 / Image des sorties n+2 bit 0
      led17 : Bool;   // output image n+2 bit 1 / Image des sorties n+2 bit 1
      led18 : Bool;   // output image n+2 bit 2 / Image des sorties n+2 bit 2
      reserved23 : Bool;
      reserved24 : Bool;
      reserved25 : Bool;
      reserved26 : Bool;
      reserved27 : Bool;
      led24 : Bool;   // output image n+3 bit 0 / Image des sorties n+3 bit 0
      led25 : Bool;   // output image n+3 bit 1 / Image des sorties n+3 bit 1
      led26 : Bool;   // output image n+3 bit 2 / Image des sorties n+3 bit 2
      reserved33 : Bool;
      reserved34 : Bool;
      reserved35 : Bool;
      reserved36 : Bool;
      reserved37 : Bool;
   END_STRUCT;
END_TYPE

TYPE "LBP_typeModularMcpUniversalInput"
TITLE = Modular MCP image / Image MCP modulaire
// Input image of universal keypad for modular MCP / Image des entrées du pupitre universel pour MCP modulaires
   STRUCT
      key0 : Bool;   // input image n+0 bit 0 / Image des entrées n+0 bit 0
      key1 : Bool;   // input image n+0 bit 1 / Image des entrées n+0 bit 1
      key2 : Bool;   // input image n+0 bit 2 / Image des entrées n+0 bit 2
      key3 : Bool;   // input image n+0 bit 3 / Image des entrées n+0 bit 3
      key4 : Bool;   // input image n+0 bit 4 / Image des entrées n+0 bit 4
      key5 : Bool;   // input image n+0 bit 5 / Image des entrées n+0 bit 5
      key6 : Bool;   // input image n+0 bit 6 / Image des entrées n+0 bit 6
      key7 : Bool;   // input image n+0 bit 7 / Image des entrées n+0 bit 7
      key8 : Bool;   // input image n+1 bit 0 / Image des entrées n+1 bit 0
      key9 : Bool;   // input image n+1 bit 1 / Image des entrées n+1 bit 1
      key10 : Bool;   // input image n+1 bit 2 / Image des entrées n+1 bit 2
      key11 : Bool;   // input image n+1 bit 3 / Image des entrées n+1 bit 3
      key12 : Bool;   // input image n+1 bit 4 / Image des entrées n+1 bit 4
      key13 : Bool;   // input image n+1 bit 5 / Image des entrées n+1 bit 5
      key14 : Bool;   // input image n+1 bit 6 / Image des entrées n+1 bit 6
      reserved17 : Bool;
      key16 : Bool;   // input image n+2 bit 0 / Image des entrées n+2 bit 0
      key17 : Bool;   // input image n+2 bit 1 / Image des entrées n+2 bit 1
      key18 : Bool;   // input image n+2 bit 2 / Image des entrées n+2 bit 2
      reserved23 : Bool;
      reserved24 : Bool;
      reserved25 : Bool;
      reserved26 : Bool;
      reserved27 : Bool;
      key24 : Bool;   // input image n+3 bit 0 / Image des entrées n+3 bit 0
      key25 : Bool;   // input image n+3 bit 1 / Image des entrées n+3 bit 1
      key26 : Bool;   // input image n+3 bit 2 / Image des entrées n+3 bit 2
      reserved33 : Bool;
      reserved34 : Bool;
      reserved35 : Bool;
      reserved36 : Bool;
      reserved37 : Bool;
   END_STRUCT;
END_TYPE

TYPE "LBP_typeModularMcpUniversalOutput"
TITLE = Modular MCP image / Image MCP modulaire
// Output image of universal keypad for modular MCP / Image des sorties du pupitre universel pour MCP modulaires
   STRUCT
      led0 : Bool;   // output image n+0 bit 0 / Image des sorties n+0 bit 0
      led1 : Bool;   // output image n+0 bit 1 / Image des sorties n+0 bit 1
      led2 : Bool;   // output image n+0 bit 2 / Image des sorties n+0 bit 2
      led3 : Bool;   // output image n+0 bit 3 / Image des sorties n+0 bit 3
      led4 : Bool;   // output image n+0 bit 4 / Image des sorties n+0 bit 4
      led5 : Bool;   // output image n+0 bit 5 / Image des sorties n+0 bit 5
      led6 : Bool;   // output image n+0 bit 6 / Image des sorties n+0 bit 6
      led7 : Bool;   // output image n+0 bit 7 / Image des sorties n+0 bit 7
      led8 : Bool;   // output image n+1 bit 0 / Image des sorties n+1 bit 0
      led9 : Bool;   // output image n+1 bit 1 / Image des sorties n+1 bit 1
      led10 : Bool;   // output image n+1 bit 2 / Image des sorties n+1 bit 2
      led11 : Bool;   // output image n+1 bit 3 / Image des sorties n+1 bit 3
      led12 : Bool;   // output image n+1 bit 4 / Image des sorties n+1 bit 4
      led13 : Bool;   // output image n+1 bit 5 / Image des sorties n+1 bit 5
      led14 : Bool;   // output image n+1 bit 6 / Image des sorties n+1 bit 6
      reserved17 : Bool;
      led16 : Bool;   // output image n+2 bit 0 / Image des sorties n+2 bit 0
      led17 : Bool;   // output image n+2 bit 1 / Image des sorties n+2 bit 1
      led18 : Bool;   // output image n+2 bit 2 / Image des sorties n+2 bit 2
      reserved23 : Bool;
      reserved24 : Bool;
      reserved25 : Bool;
      reserved26 : Bool;
      reserved27 : Bool;
      led24 : Bool;   // output image n+3 bit 0 / Image des sorties n+3 bit 0
      led25 : Bool;   // output image n+3 bit 1 / Image des sorties n+3 bit 1
      led26 : Bool;   // output image n+3 bit 2 / Image des sorties n+3 bit 2
      reserved33 : Bool;
      reserved34 : Bool;
      reserved35 : Bool;
      reserved36 : Bool;
      reserved37 : Bool;
   END_STRUCT;
END_TYPE

TYPE "LBP_typePowerrideConfig"
TITLE = Data type for configuration of Powerride / Type de données pour la configuration Powerride
// User data type for LBP_PowerrideConfig / Type de données utilisateur pour LBP_PowerrideConfig
   STRUCT
      pos100 { S7_SetPoint := 'True'} : USInt := 0;   // [1..36] switch position at 100% ovr / [1..36] position du commutateur à correction 100 %
      posMax { S7_SetPoint := 'True'} : USInt := 0;   // [1..36] switch position at maximum ovr / [1..36] position du commutateur à correction maximale
      delay100 { S7_SetPoint := 'True'} : Time := T#500MS;   // time delay at 100% before continuing ovr / délai à 100 % avant de continuer correction
      switchPos { S7_SetPoint := 'True'} : Array[1..36] of "LBP_typePowerrideConfigPos";   // value, colour and vibration for position / valeur, couleur et vibration pour la position
   END_STRUCT;
END_TYPE

TYPE "LBP_typePowerrideConfigPos"
TITLE = Data type for configuration of a Powerride position / Type de données pour configuration d'une position Powerride
// User data type for LBP_PowerrideConfig (sub type) / Type de données utilisateur pour LBP_PowerrideConfig (sous-type)
   STRUCT
      value { S7_SetPoint := 'True'} : USInt;   // override factor / facteur de correction
      ledColor { S7_SetPoint := 'True'} : USInt;   // color of scale LEDs / couleur des LED d'échelle
      vibrationIndex { S7_SetPoint := 'True'} : USInt;   // index of vibration pattern / indice du modèle de vibration
   END_STRUCT;
END_TYPE

TYPE "LBP_typePowerrideInput"
TITLE = Powerride image / Image Powerride
// Input image of powerride / Image des entrées de Powerride
   STRUCT
      pushButton : Bool;   // true, when push button pressed / vrai, lorsque le bouton-poussoir est enfoncé
      reserved01 : Bool;
      reserved02 : Bool;
      reserved03 : Bool;
      reserved04 : Bool;
      reserved05 : Bool;
      reserved06 : Bool;
      reserved07 : Bool;
      powerrideCounter : USInt;   // [0..255] Override switch position / [0..255] Corriger la position du commutateur
   END_STRUCT;
END_TYPE

TYPE "LBP_typePowerrideOutput"
TITLE = Powerride image / Image Powerride
// Output image of powerride / Image des sorties de Powerride
   STRUCT
      ledInfo : DWord;   // Led24..Led0
      scaleRed : Bool;   // when true, red scale LED is on / si vrai, la LED d'échelle rouge est allumée
      scaleGreen : Bool;   // when true, green scale LED is on / si vrai, la LED d'échelle verte est allumée
      scaleBlue : Bool;   // when true, blue scale LED ist on / si vrai, la LED d'échelle bleue est allumée
      buttonRed : Bool;   // when true, red push button LED is on / si vrai, la LED rouge du bouton-poussoir est allumée
      buttonGreen : Bool;   // when true, green push button LED is on / si vrai, la LED verte du bouton-poussoir est allumée
      buttonBlue : Bool;   // when true, blue push button LED is on / Si TRUE, la LED bleue du bouton-poussoir est allumée
      reserved46 : Bool;
      reserved47 : Bool;
      vibrationPattern : USInt;   // vibration pattern index to be used / indice du modèle de vibration à utiliser
   END_STRUCT;
END_TYPE

TYPE "LBP_typeNCVariableToken"
TITLE = LBP_ReadVar and LBP_WriteVar Input Interface / Interface d'entrée LBP_ReadVar et LBP_WriteVar
// User Data Type for LBP_ReadVar[FB2] and LBP_WriteVar[FB3] Input Parameter Addrx / Type de données utilisateur pour les paramètres d'entrée Addrx LBP_ReadVar[FB2] et LBP_WriteVar[FB3]
   STRUCT
      syntaxId : Byte;   // syntax ID / ID de syntaxe
      areaAndUnit : Byte;   // area and unit / zone et unité
      column : Word;   // column / colonne
      row : Word;   // row / ligne
      blockType : Byte;   // block type / type de bloc
      numberOfRows : Byte;   // number of rows / nombre de lignes
      dataTypeCode : Byte;   // data type code / code de type de données
      length : Byte;   // length of data type / longueur de type de données
   END_STRUCT;
END_TYPE

TYPE "LBP_typeNCVariableTokenBool"
TITLE = LBP_ReadVar and LBP_WriteVar Interface / Interface LBP_ReadVar et LBP_WriteVar
// User Data Type for LBP_ReadVar[FB2] and LBP_WriteVar[FB3] Parameters / Type de données utilisateur pour les paramètres LBP_ReadVar[FB2] et LBP_WriteVar[FB3]
   STRUCT
      token : "LBP_typeNCVariableToken";   // User Data Type for LBP_ReadVar[FB2] and LBP_WriteVar[FB3] Input Parameter Addrx / Type de données utilisateur pour les paramètres d'entrée Addrx LBP_ReadVar[FB2] et LBP_WriteVar[FB3]
      value : Bool;   // Data Type for LBP_ReadVar[FB2] and LBP_WriteVar[FB3] InOut Parameter SDx / Type de données pour les paramètres E/S SDx LBP_ReadVar[FB2] et LBP_WriteVar[FB3]
   END_STRUCT;
END_TYPE

TYPE "LBP_typeNCVariableTokenDInt"
TITLE = LBP_ReadVar and LBP_WriteVar Interface / Interface LBP_ReadVar et LBP_WriteVar
// User Data Type for LBP_ReadVar[FB2] and LBP_WriteVar[FB3] Parameters / Type de données utilisateur pour les paramètres LBP_ReadVar[FB2] et LBP_WriteVar[FB3]
   STRUCT
      token : "LBP_typeNCVariableToken";   // User Data Type for LBP_ReadVar[FB2] and LBP_WriteVar[FB3] Input Parameter Addrx / Type de données utilisateur pour les paramètres d'entrée Addrx LBP_ReadVar[FB2] et LBP_WriteVar[FB3]
      value : DInt;   // Data Type for LBP_ReadVar[FB2] and LBP_WriteVar[FB3] InOut Parameter SDx / Type de données pour les paramètres E/S SDx LBP_ReadVar[FB2] et LBP_WriteVar[FB3]
   END_STRUCT;
END_TYPE

